LIN {X -0.022,Y -551.282,Z 288.033,A 0.000,B 0.000,C 90.000,E1 221.881} C_DIS
LIN {X -0.166,Y -545.235,Z 288.022,A 0.000,B 0.000,C 90.000,E1 219.930} C_DIS
LIN {X -0.082,Y -540.917,Z 288.014,A 0.000,B 0.000,C 90.000,E1 218.508} C_DIS
LIN {X 0.010,Y -536.637,Z 288.006,A 0.000,B 0.000,C 90.000,E1 217.076} C_DIS
LIN {X -0.298,Y -530.712,Z 287.995,A 0.000,B 0.000,C 90.000,E1 215.105} C_DIS
LIN {X 0.124,Y -524.882,Z 287.984,A 0.000,B 0.000,C 90.000,E1 213.038} C_DIS
LIN {X 0.156,Y -517.882,Z 287.969,A 0.000,B 0.000,C 90.000,E1 210.413} C_DIS
LIN {X -0.211,Y -511.936,Z 287.956,A 0.000,B 0.000,C 90.000,E1 208.103} C_DIS
LIN {X -0.005,Y -505.662,Z 287.941,A 0.000,B 0.000,C 90.000,E1 205.412} C_DIS
LIN {X -0.124,Y -501.187,Z 287.930,A 0.000,B 0.000,C 90.000,E1 203.334} C_DIS
LIN {X -0.097,Y -496.953,Z 287.918,A 0.000,B 0.000,C 90.000,E1 201.227} C_DIS
LIN {X 0.055,Y -493.512,Z 287.908,A 0.000,B 0.000,C 90.000,E1 199.396} C_DIS
LIN {X -0.125,Y -489.341,Z 287.894,A 0.000,B 0.000,C 90.000,E1 196.985} C_DIS
LIN {X -0.107,Y -485.490,Z 287.881,A 0.000,B 0.000,C 90.000,E1 194.537} C_DIS
LIN {X 0.015,Y -482.002,Z 287.867,A 0.000,B 0.000,C 90.000,E1 192.063} C_DIS
LIN {X -0.021,Y -479.203,Z 287.855,A 0.000,B 0.000,C 90.000,E1 189.905} C_DIS
LIN {X -0.211,Y -476.723,Z 287.843,A 0.000,B 0.000,C 90.000,E1 187.757} C_DIS
LIN {X 0.179,Y -474.137,Z 287.829,A 0.000,B 0.000,C 90.000,E1 185.220} C_DIS
LIN {X 0.182,Y -471.554,Z 287.814,A 0.000,B 0.000,C 90.000,E1 182.407} C_DIS
LIN {X 0.049,Y -469.852,Z 287.801,A 0.000,B 0.000,C 90.000,E1 180.229} C_DIS
LIN {X -0.125,Y -468.633,Z 287.789,A 0.000,B 0.000,C 90.000,E1 178.051} C_DIS
LIN {X 0.163,Y -467.261,Z 287.770,A 0.000,B 0.000,C 90.000,E1 174.552} C_DIS
LIN {X 0.067,Y -466.887,Z 287.758,A 0.000,B 0.000,C 90.000,E1 172.356} C_DIS
LIN {X 0.114,Y -466.574,Z 287.742,A 0.000,B 0.000,C 90.000,E1 169.511} C_DIS
LIN {X -0.130,Y -466.836,Z 287.726,A 0.000,B 0.000,C 90.000,E1 166.700} C_DIS
LIN {X 0.160,Y -468.096,Z 287.707,A 0.000,B 0.000,C 90.000,E1 163.196} C_DIS
LIN {X 0.075,Y -470.064,Z 287.689,A 0.000,B 0.000,C 90.000,E1 160.061} C_DIS
LIN {X 0.258,Y -471.526,Z 287.679,A 0.000,B 0.000,C 90.000,E1 158.156} C_DIS
LIN {X 0.123,Y -474.366,Z 287.663,A 0.000,B 0.000,C 90.000,E1 155.357} C_DIS
LIN {X -0.198,Y -478.123,Z 287.646,A 0.000,B 0.000,C 90.000,E1 152.281} C_DIS
LIN {X 0.097,Y -481.402,Z 287.634,A 0.000,B 0.000,C 90.000,E1 150.078} C_DIS
LIN {X 0.128,Y -484.933,Z 287.622,A 0.000,B 0.000,C 90.000,E1 147.916} C_DIS
LIN {X -0.149,Y -488.614,Z 287.610,A 0.000,B 0.000,C 90.000,E1 145.801} C_DIS
LIN {X -0.316,Y -491.783,Z 287.600,A 0.000,B 0.000,C 90.000,E1 143.989} C_DIS
LIN {X 0.172,Y -494.913,Z 287.590,A 0.000,B 0.000,C 90.000,E1 142.110} C_DIS
LIN {X -0.080,Y -496.875,Z 287.583,A 0.000,B 0.000,C 90.000,E1 140.928} C_DIS
LIN {X 0.076,Y -498.689,Z 287.576,A 0.000,B 0.000,C 90.000,E1 139.703} C_DIS
LIN {X 0.195,Y -500.322,Z 287.570,A 0.000,B 0.000,C 90.000,E1 138.485} C_DIS
LIN {X -0.034,Y -501.602,Z 287.563,A 0.000,B 0.000,C 90.000,E1 137.310} C_DIS
LIN {X 0.042,Y -502.103,Z 287.560,A 0.000,B 0.000,C 90.000,E1 136.701} C_DIS
LIN {X -0.028,Y -502.598,Z 287.555,A 0.000,B 0.000,C 90.000,E1 135.810} C_DIS
LIN {X -0.091,Y -502.898,Z 287.550,A 0.000,B 0.000,C 90.000,E1 134.919} C_DIS
LIN {X 0.067,Y -502.896,Z 287.543,A 0.000,B 0.000,C 90.000,E1 133.704} C_DIS
LIN {X 0.001,Y -502.579,Z 287.538,A 0.000,B 0.000,C 90.000,E1 132.813} C_DIS
LIN {X -0.038,Y -502.029,Z 287.533,A 0.000,B 0.000,C 90.000,E1 131.919} C_DIS
LIN {X 0.129,Y -500.892,Z 287.526,A 0.000,B 0.000,C 90.000,E1 130.701} C_DIS
LIN {X 0.081,Y -499.879,Z 287.521,A 0.000,B 0.000,C 90.000,E1 129.806} C_DIS
LIN {X -0.104,Y -498.289,Z 287.515,A 0.000,B 0.000,C 90.000,E1 128.624} C_DIS
LIN {X 0.078,Y -496.609,Z 287.508,A 0.000,B 0.000,C 90.000,E1 127.397} C_DIS
LIN {X -0.165,Y -494.765,Z 287.501,A 0.000,B 0.000,C 90.000,E1 126.217} C_DIS
LIN {X -0.078,Y -492.159,Z 287.493,A 0.000,B 0.000,C 90.000,E1 124.692} C_DIS
LIN {X -0.037,Y -489.306,Z 287.484,A 0.000,B 0.000,C 90.000,E1 123.166} C_DIS
LIN {X -0.082,Y -485.832,Z 287.474,A 0.000,B 0.000,C 90.000,E1 121.337} C_DIS
LIN {X -0.241,Y -483.532,Z 287.467,A 0.000,B 0.000,C 90.000,E1 120.129} C_DIS
LIN {X -0.277,Y -479.342,Z 287.455,A 0.000,B 0.000,C 90.000,E1 117.975} C_DIS
LIN {X -0.162,Y -476.366,Z 287.447,A 0.000,B 0.000,C 90.000,E1 116.411} C_DIS
LIN {X -0.068,Y -473.881,Z 287.440,A 0.000,B 0.000,C 90.000,E1 115.155} C_DIS
LIN {X -0.004,Y -471.585,Z 287.433,A 0.000,B 0.000,C 90.000,E1 113.898} C_DIS
LIN {X -0.174,Y -466.921,Z 287.419,A 0.000,B 0.000,C 90.000,E1 111.408} C_DIS
LIN {X -0.099,Y -463.544,Z 287.408,A 0.000,B 0.000,C 90.000,E1 109.504} C_DIS
LIN {X -0.105,Y -460.881,Z 287.400,A 0.000,B 0.000,C 90.000,E1 107.928} C_DIS
LIN {X -0.145,Y -460.875,Z 287.400,A 0.000,B 0.000,C 90.000,E1 107.928} C_DIS
LIN {X -0.237,Y -467.713,Z 287.383,A 0.000,B 0.000,C 90.000,E1 104.954} C_DIS
LIN {X 0.187,Y -475.922,Z 287.357,A 0.000,B 0.000,C 90.000,E1 100.197} C_DIS
LIN {X 0.027,Y -476.358,Z 287.355,A 0.000,B 0.000,C 90.000,E1 99.905} C_DIS
LIN {X -0.017,Y -481.880,Z 287.331,A 0.000,B 0.000,C 90.000,E1 95.568} C_DIS
LIN {X -0.170,Y -482.194,Z 287.329,A 0.000,B 0.000,C 90.000,E1 95.277} C_DIS
LIN {X -0.236,Y -485.368,Z 287.305,A 0.000,B 0.000,C 90.000,E1 90.974} C_DIS
LIN {X 0.073,Y -485.531,Z 287.304,A 0.000,B 0.000,C 90.000,E1 90.630} C_DIS
LIN {X -0.204,Y -486.347,Z 287.281,A 0.000,B 0.000,C 90.000,E1 86.674} C_DIS
LIN {X 0.106,Y -486.369,Z 287.280,A 0.000,B 0.000,C 90.000,E1 86.331} C_DIS
LIN {X -0.212,Y -486.061,Z 287.276,A 0.000,B 0.000,C 90.000,E1 85.755} C_DIS
LIN {X 0.130,Y -484.693,Z 287.254,A 0.000,B 0.000,C 90.000,E1 81.724} C_DIS
LIN {X -0.002,Y -484.531,Z 287.252,A 0.000,B 0.000,C 90.000,E1 81.432} C_DIS
LIN {X -0.132,Y -480.469,Z 287.227,A 0.000,B 0.000,C 90.000,E1 76.825} C_DIS
LIN {X -0.235,Y -474.228,Z 287.201,A 0.000,B 0.000,C 90.000,E1 72.181} C_DIS
LIN {X 0.183,Y -473.729,Z 287.199,A 0.000,B 0.000,C 90.000,E1 71.819} C_DIS
LIN {X 0.081,Y -472.855,Z 287.197,A 0.000,B 0.000,C 90.000,E1 71.402} C_DIS
LIN {X 0.041,Y -472.855,Z 287.197,A 0.000,B 0.000,C 90.000,E1 71.402} C_DIS
LIN {X 0.283,Y -476.430,Z 287.189,A 0.000,B 0.000,C 90.000,E1 69.934} C_DIS
LIN {X 0.008,Y -482.896,Z 287.175,A 0.000,B 0.000,C 90.000,E1 67.486} C_DIS
LIN {X -0.165,Y -489.519,Z 287.161,A 0.000,B 0.000,C 90.000,E1 65.049} C_DIS
LIN {X -0.053,Y -493.811,Z 287.153,A 0.000,B 0.000,C 90.000,E1 63.512} C_DIS
LIN {X -0.125,Y -500.706,Z 287.139,A 0.000,B 0.000,C 90.000,E1 61.101} C_DIS
LIN {X 0.059,Y -505.947,Z 287.129,A 0.000,B 0.000,C 90.000,E1 59.282} C_DIS
LIN {X 0.070,Y -512.082,Z 287.118,A 0.000,B 0.000,C 90.000,E1 57.199} C_DIS
LIN {X 0.086,Y -516.294,Z 287.110,A 0.000,B 0.000,C 90.000,E1 55.722} C_DIS
LIN {X -0.049,Y -519.604,Z 287.103,A 0.000,B 0.000,C 90.000,E1 54.562} C_DIS
LIN {X -0.263,Y -522.649,Z 287.097,A 0.000,B 0.000,C 90.000,E1 53.417} C_DIS
LIN {X 0.304,Y -525.486,Z 287.090,A 0.000,B 0.000,C 90.000,E1 52.190} C_DIS
LIN {X 0.203,Y -527.474,Z 287.085,A 0.000,B 0.000,C 90.000,E1 51.331} C_DIS
LIN {X 0.020,Y -529.949,Z 287.079,A 0.000,B 0.000,C 90.000,E1 50.194} C_DIS
LIN {X 0.301,Y -531.668,Z 287.074,A 0.000,B 0.000,C 90.000,E1 49.299} C_DIS
LIN {X -0.155,Y -533.178,Z 287.069,A 0.000,B 0.000,C 90.000,E1 48.485} C_DIS
LIN {X 0.102,Y -534.990,Z 287.063,A 0.000,B 0.000,C 90.000,E1 47.310} C_DIS
LIN {X 0.001,Y -536.441,Z 287.057,A 0.000,B 0.000,C 90.000,E1 46.176} C_DIS
LIN {X -0.070,Y -537.575,Z 287.050,A 0.000,B 0.000,C 90.000,E1 45.040} C_DIS
LIN {X 0.246,Y -538.429,Z 287.044,A 0.000,B 0.000,C 90.000,E1 43.866} C_DIS
LIN {X -0.179,Y -539.008,Z 287.038,A 0.000,B 0.000,C 90.000,E1 42.771} C_DIS
LIN {X 0.163,Y -539.340,Z 287.031,A 0.000,B 0.000,C 90.000,E1 41.595} C_DIS
LIN {X 0.149,Y -539.479,Z 287.025,A 0.000,B 0.000,C 90.000,E1 40.458} C_DIS
LIN {X -0.209,Y -539.367,Z 287.019,A 0.000,B 0.000,C 90.000,E1 39.358} C_DIS
LIN {X 0.209,Y -538.800,Z 287.011,A 0.000,B 0.000,C 90.000,E1 37.890} C_DIS
LIN {X -0.148,Y -537.903,Z 287.003,A 0.000,B 0.000,C 90.000,E1 36.503} C_DIS
LIN {X -0.107,Y -537.027,Z 286.996,A 0.000,B 0.000,C 90.000,E1 35.358} C_DIS
LIN {X 0.051,Y -535.988,Z 286.990,A 0.000,B 0.000,C 90.000,E1 34.199} C_DIS
LIN {X 0.193,Y -534.349,Z 286.981,A 0.000,B 0.000,C 90.000,E1 32.467} C_DIS
LIN {X -0.277,Y -532.519,Z 286.971,A 0.000,B 0.000,C 90.000,E1 30.797} C_DIS
LIN {X 0.141,Y -530.682,Z 286.961,A 0.000,B 0.000,C 90.000,E1 29.027} C_DIS
LIN {X 0.046,Y -528.801,Z 286.952,A 0.000,B 0.000,C 90.000,E1 27.308} C_DIS
LIN {X -0.114,Y -526.875,Z 286.942,A 0.000,B 0.000,C 90.000,E1 25.591} C_DIS
LIN {X 0.165,Y -525.172,Z 286.932,A 0.000,B 0.000,C 90.000,E1 23.823} C_DIS
LIN {X 0.157,Y -523.230,Z 286.921,A 0.000,B 0.000,C 90.000,E1 21.791} C_DIS
LIN {X -0.022,Y -521.984,Z 286.913,A 0.000,B 0.000,C 90.000,E1 20.355} C_DIS
LIN {X -0.103,Y -520.900,Z 286.905,A 0.000,B 0.000,C 90.000,E1 18.906} C_DIS
LIN {X -0.060,Y -519.660,Z 286.895,A 0.000,B 0.000,C 90.000,E1 17.149} C_DIS
LIN {X -0.251,Y -518.083,Z 286.881,A 0.000,B 0.000,C 90.000,E1 14.537} C_DIS
LIN {X -0.203,Y -517.233,Z 286.869,A 0.000,B 0.000,C 90.000,E1 12.479} C_DIS
LIN {X 0.189,Y -516.314,Z 286.853,A 0.000,B 0.000,C 90.000,E1 9.500} C_DIS
LIN {X -0.015,Y -516.024,Z 286.842,A 0.000,B 0.000,C 90.000,E1 7.466} C_DIS
LIN {X 0.141,Y -516.118,Z 286.830,A 0.000,B 0.000,C 90.000,E1 5.391} C_DIS
LIN {X -0.225,Y -516.505,Z 286.820,A 0.000,B 0.000,C 90.000,E1 3.669} C_DIS
LIN {X 0.127,Y -517.693,Z 286.802,A 0.000,B 0.000,C 90.000,E1 0.401} C_DIS
LIN {X -0.102,Y -519.014,Z 286.791,A 0.000,B 0.000,C 90.000,E1 358.339} C_DIS
LIN {X 0.061,Y -520.698,Z 286.779,A 0.000,B 0.000,C 90.000,E1 356.274} C_DIS
LIN {X 0.248,Y -523.662,Z 286.763,A 0.000,B 0.000,C 90.000,E1 353.337} C_DIS
LIN {X 0.219,Y -528.870,Z 286.744,A 0.000,B 0.000,C 90.000,E1 349.859} C_DIS
LIN {X -0.151,Y -533.012,Z 286.733,A 0.000,B 0.000,C 90.000,E1 347.881} C_DIS
LIN {X -0.010,Y -538.644,Z 286.720,A 0.000,B 0.000,C 90.000,E1 345.574} C_DIS
LIN {X 0.005,Y -542.943,Z 286.710,A 0.000,B 0.000,C 90.000,E1 343.866} C_DIS
LIN {X 0.036,Y -550.760,Z 286.695,A 0.000,B 0.000,C 90.000,E1 341.040} C_DIS
LIN {X 0.290,Y -561.382,Z 286.676,A 0.000,B 0.000,C 90.000,E1 337.667} C_DIS
LIN {X 0.104,Y -566.038,Z 286.668,A 0.000,B 0.000,C 90.000,E1 336.305} C_DIS
LIN {X 0.063,Y -568.796,Z 286.664,A 0.000,B 0.000,C 90.000,E1 335.485} C_DIS
LIN {X -0.284,Y -573.663,Z 286.656,A 0.000,B 0.000,C 90.000,E1 334.152} C_DIS
LIN {X 0.224,Y -578.648,Z 286.649,A 0.000,B 0.000,C 90.000,E1 332.743} C_DIS
LIN {X 0.175,Y -584.349,Z 286.640,A 0.000,B 0.000,C 90.000,E1 331.129} C_DIS
LIN {X 0.078,Y -587.101,Z 286.635,A 0.000,B 0.000,C 90.000,E1 330.333} C_DIS
LIN {X 0.173,Y -593.390,Z 286.625,A 0.000,B 0.000,C 90.000,E1 328.456} C_DIS
LIN {X -0.085,Y -599.852,Z 286.615,A 0.000,B 0.000,C 90.000,E1 326.628} C_DIS
LIN {X 0.137,Y -606.584,Z 286.604,A 0.000,B 0.000,C 90.000,E1 324.769} C_DIS
LIN {X -0.200,Y -611.352,Z 286.597,A 0.000,B 0.000,C 90.000,E1 323.497} C_DIS
LIN {X 0.098,Y -614.969,Z 286.591,A 0.000,B 0.000,C 90.000,E1 322.431} C_DIS
LIN {X -0.043,Y -618.442,Z 286.586,A 0.000,B 0.000,C 90.000,E1 321.412} C_DIS
LIN {X 0.022,Y -623.383,Z 286.577,A 0.000,B 0.000,C 90.000,E1 319.865} C_DIS
LIN {X 0.117,Y -628.029,Z 286.569,A 0.000,B 0.000,C 90.000,E1 318.324} C_DIS
LIN {X 0.083,Y -630.918,Z 286.563,A 0.000,B 0.000,C 90.000,E1 317.310} C_DIS
LIN {X -0.125,Y -635.283,Z 286.555,A 0.000,B 0.000,C 90.000,E1 315.810} C_DIS
LIN {X 0.290,Y -638.880,Z 286.547,A 0.000,B 0.000,C 90.000,E1 314.514} C_DIS
LIN {X -0.145,Y -642.391,Z 286.541,A 0.000,B 0.000,C 90.000,E1 313.299} C_DIS
LIN {X 0.088,Y -644.386,Z 286.536,A 0.000,B 0.000,C 90.000,E1 312.528} C_DIS
LIN {X 0.272,Y -646.963,Z 286.531,A 0.000,B 0.000,C 90.000,E1 311.515} C_DIS
LIN {X 0.060,Y -649.243,Z 286.525,A 0.000,B 0.000,C 90.000,E1 310.539} C_DIS
LIN {X -0.120,Y -651.334,Z 286.520,A 0.000,B 0.000,C 90.000,E1 309.564} C_DIS
LIN {X -0.298,Y -654.019,Z 286.512,A 0.000,B 0.000,C 90.000,E1 308.096} C_DIS
LIN {X 0.088,Y -655.509,Z 286.506,A 0.000,B 0.000,C 90.000,E1 307.076} C_DIS
LIN {X 0.102,Y -656.775,Z 286.501,A 0.000,B 0.000,C 90.000,E1 306.091} C_DIS
LIN {X 0.116,Y -657.281,Z 286.498,A 0.000,B 0.000,C 90.000,E1 305.598} C_DIS
LIN {X 0.154,Y -657.718,Z 286.492,A 0.000,B 0.000,C 90.000,E1 304.612} C_DIS
LIN {X 0.191,Y -657.885,Z 286.487,A 0.000,B 0.000,C 90.000,E1 303.627} C_DIS
LIN {X 0.310,Y -657.889,Z 286.483,A 0.000,B 0.000,C 90.000,E1 302.880} C_DIS
LIN {X 0.080,Y -657.516,Z 286.479,A 0.000,B 0.000,C 90.000,E1 302.163} C_DIS
LIN {X 0.091,Y -657.134,Z 286.476,A 0.000,B 0.000,C 90.000,E1 301.671} C_DIS
LIN {X 0.203,Y -656.212,Z 286.472,A 0.000,B 0.000,C 90.000,E1 300.924} C_DIS
LIN {X -0.030,Y -654.993,Z 286.468,A 0.000,B 0.000,C 90.000,E1 300.207} C_DIS
LIN {X 0.160,Y -652.992,Z 286.462,A 0.000,B 0.000,C 90.000,E1 299.205} C_DIS
LIN {X 0.001,Y -650.651,Z 286.457,A 0.000,B 0.000,C 90.000,E1 298.231} C_DIS
LIN {X -0.280,Y -648.844,Z 286.453,A 0.000,B 0.000,C 90.000,E1 297.513} C_DIS
LIN {X 0.170,Y -645.743,Z 286.446,A 0.000,B 0.000,C 90.000,E1 296.232} C_DIS
LIN {X -0.221,Y -641.747,Z 286.438,A 0.000,B 0.000,C 90.000,E1 294.771} C_DIS
LIN {X -0.166,Y -638.308,Z 286.431,A 0.000,B 0.000,C 90.000,E1 293.515} C_DIS
LIN {X -0.217,Y -635.664,Z 286.425,A 0.000,B 0.000,C 90.000,E1 292.514} C_DIS
LIN {X -0.102,Y -631.085,Z 286.415,A 0.000,B 0.000,C 90.000,E1 290.737} C_DIS
LIN {X -0.304,Y -625.969,Z 286.404,A 0.000,B 0.000,C 90.000,E1 288.725} C_DIS
LIN {X -0.035,Y -621.828,Z 286.394,A 0.000,B 0.000,C 90.000,E1 286.913} C_DIS
LIN {X 0.083,Y -617.059,Z 286.381,A 0.000,B 0.000,C 90.000,E1 284.592} C_DIS
LIN {X -0.023,Y -611.498,Z 286.362,A 0.000,B 0.000,C 90.000,E1 281.243} C_DIS
LIN {X 0.188,Y -608.186,Z 286.348,A 0.000,B 0.000,C 90.000,E1 278.624} C_DIS
LIN {X -0.246,Y -605.664,Z 286.332,A 0.000,B 0.000,C 90.000,E1 275.796} C_DIS
LIN {X -0.110,Y -604.050,Z 286.312,A 0.000,B 0.000,C 90.000,E1 272.121} C_DIS
LIN {X -0.009,Y -603.945,Z 286.294,A 0.000,B 0.000,C 90.000,E1 268.969} C_DIS
LIN {X -0.193,Y -605.476,Z 286.275,A 0.000,B 0.000,C 90.000,E1 265.584} C_DIS
LIN {X 0.194,Y -607.166,Z 286.264,A 0.000,B 0.000,C 90.000,E1 263.457} C_DIS
LIN {X 0.232,Y -610.043,Z 286.249,A 0.000,B 0.000,C 90.000,E1 260.849} C_DIS
LIN {X 0.136,Y -613.319,Z 286.236,A 0.000,B 0.000,C 90.000,E1 258.522} C_DIS
LIN {X 0.252,Y -616.132,Z 286.226,A 0.000,B 0.000,C 90.000,E1 256.700} C_DIS
LIN {X -0.173,Y -618.906,Z 286.216,A 0.000,B 0.000,C 90.000,E1 254.936} C_DIS
LIN {X -0.092,Y -619.987,Z 286.212,A 0.000,B 0.000,C 90.000,E1 254.157} C_DIS
LIN {X 0.005,Y -620.838,Z 286.208,A 0.000,B 0.000,C 90.000,E1 253.378} C_DIS
LIN {X 0.113,Y -621.447,Z 286.203,A 0.000,B 0.000,C 90.000,E1 252.598} C_DIS
LIN {X -0.248,Y -622.517,Z 286.195,A 0.000,B 0.000,C 90.000,E1 251.094} C_DIS
LIN {X -0.149,Y -622.786,Z 286.189,A 0.000,B 0.000,C 90.000,E1 250.061} C_DIS
LIN {X 0.181,Y -622.785,Z 286.185,A 0.000,B 0.000,C 90.000,E1 249.263} C_DIS
LIN {X -0.303,Y -622.345,Z 286.179,A 0.000,B 0.000,C 90.000,E1 248.284} C_DIS
LIN {X 0.019,Y -621.839,Z 286.175,A 0.000,B 0.000,C 90.000,E1 247.486} C_DIS
LIN {X -0.240,Y -621.023,Z 286.171,A 0.000,B 0.000,C 90.000,E1 246.741} C_DIS
LIN {X 0.301,Y -619.565,Z 286.165,A 0.000,B 0.000,C 90.000,E1 245.665} C_DIS
LIN {X 0.016,Y -618.228,Z 286.161,A 0.000,B 0.000,C 90.000,E1 244.921} C_DIS
LIN {X -0.038,Y -616.106,Z 286.155,A 0.000,B 0.000,C 90.000,E1 243.896} C_DIS
LIN {X -0.142,Y -613.014,Z 286.148,A 0.000,B 0.000,C 90.000,E1 242.615} C_DIS
LIN {X -0.015,Y -609.650,Z 286.141,A 0.000,B 0.000,C 90.000,E1 241.307} C_DIS
LIN {X 0.056,Y -606.046,Z 286.133,A 0.000,B 0.000,C 90.000,E1 239.999} C_DIS
LIN {X 0.120,Y -603.094,Z 286.128,A 0.000,B 0.000,C 90.000,E1 238.948} C_DIS
LIN {X 0.095,Y -598.460,Z 286.119,A 0.000,B 0.000,C 90.000,E1 237.375} C_DIS
LIN {X -0.239,Y -594.425,Z 286.112,A 0.000,B 0.000,C 90.000,E1 236.087} C_DIS
LIN {X 0.296,Y -591.080,Z 286.106,A 0.000,B 0.000,C 90.000,E1 234.975} C_DIS
LIN {X -0.124,Y -585.783,Z 286.097,A 0.000,B 0.000,C 90.000,E1 233.417} C_DIS
LIN {X -0.121,Y -579.944,Z 286.086,A 0.000,B 0.000,C 90.000,E1 231.537} C_DIS
LIN {X 0.084,Y -576.555,Z 286.080,A 0.000,B 0.000,C 90.000,E1 230.436} C_DIS
LIN {X 0.273,Y -569.783,Z 286.068,A 0.000,B 0.000,C 90.000,E1 228.243} C_DIS
LIN {X -0.035,Y -565.590,Z 286.061,A 0.000,B 0.000,C 90.000,E1 226.905} C_DIS
LIN {X 0.059,Y -560.458,Z 286.051,A 0.000,B 0.000,C 90.000,E1 225.243} C_DIS
LIN {X 0.043,Y -555.295,Z 286.042,A 0.000,B 0.000,C 90.000,E1 223.581} C_DIS
LIN {X -0.081,Y -550.166,Z 286.033,A 0.000,B 0.000,C 90.000,E1 221.919} C_DIS
LIN {X 0.112,Y -544.110,Z 286.022,A 0.000,B 0.000,C 90.000,E1 219.930} C_DIS
LIN {X -0.162,Y -539.773,Z 286.014,A 0.000,B 0.000,C 90.000,E1 218.543} C_DIS
LIN {X 0.243,Y -535.494,Z 286.006,A 0.000,B 0.000,C 90.000,E1 217.076} C_DIS
LIN {X -0.096,Y -529.555,Z 285.995,A 0.000,B 0.000,C 90.000,E1 215.105} C_DIS
LIN {X -0.145,Y -523.735,Z 285.984,A 0.000,B 0.000,C 90.000,E1 213.086} C_DIS
LIN {X 0.178,Y -517.508,Z 285.971,A 0.000,B 0.000,C 90.000,E1 210.718} C_DIS
LIN {X -0.117,Y -510.755,Z 285.956,A 0.000,B 0.000,C 90.000,E1 208.103} C_DIS
LIN {X 0.049,Y -504.490,Z 285.941,A 0.000,B 0.000,C 90.000,E1 205.412} C_DIS
LIN {X -0.173,Y -500.627,Z 285.931,A 0.000,B 0.000,C 90.000,E1 203.643} C_DIS
LIN {X -0.222,Y -496.967,Z 285.921,A 0.000,B 0.000,C 90.000,E1 201.844} C_DIS
LIN {X 0.023,Y -492.365,Z 285.908,A 0.000,B 0.000,C 90.000,E1 199.396} C_DIS
LIN {X -0.175,Y -487.682,Z 285.893,A 0.000,B 0.000,C 90.000,E1 196.677} C_DIS
LIN {X -0.206,Y -484.341,Z 285.881,A 0.000,B 0.000,C 90.000,E1 194.537} C_DIS
LIN {X 0.159,Y -481.701,Z 285.870,A 0.000,B 0.000,C 90.000,E1 192.647} C_DIS
LIN {X 0.112,Y -478.889,Z 285.858,A 0.000,B 0.000,C 90.000,E1 190.489} C_DIS
LIN {X -0.238,Y -475.986,Z 285.845,A 0.000,B 0.000,C 90.000,E1 188.049} C_DIS
LIN {X 0.137,Y -473.403,Z 285.831,A 0.000,B 0.000,C 90.000,E1 185.511} C_DIS
LIN {X 0.152,Y -470.823,Z 285.815,A 0.000,B 0.000,C 90.000,E1 182.694} C_DIS
LIN {X -0.231,Y -468.922,Z 285.801,A 0.000,B 0.000,C 90.000,E1 180.229} C_DIS
LIN {X 0.040,Y -467.675,Z 285.789,A 0.000,B 0.000,C 90.000,E1 177.993} C_DIS
LIN {X -0.150,Y -466.533,Z 285.773,A 0.000,B 0.000,C 90.000,E1 175.179} C_DIS
LIN {X -0.101,Y -466.011,Z 285.759,A 0.000,B 0.000,C 90.000,E1 172.648} C_DIS
LIN {X 0.107,Y -465.735,Z 285.745,A 0.000,B 0.000,C 90.000,E1 170.095} C_DIS
LIN {X 0.094,Y -465.947,Z 285.728,A 0.000,B 0.000,C 90.000,E1 166.937} C_DIS
LIN {X -0.234,Y -467.081,Z 285.708,A 0.000,B 0.000,C 90.000,E1 163.504} C_DIS
LIN {X 0.074,Y -469.009,Z 285.691,A 0.000,B 0.000,C 90.000,E1 160.315} C_DIS
LIN {X 0.180,Y -470.706,Z 285.679,A 0.000,B 0.000,C 90.000,E1 158.103} C_DIS
LIN {X 0.007,Y -473.564,Z 285.663,A 0.000,B 0.000,C 90.000,E1 155.305} C_DIS
LIN {X 0.028,Y -478.249,Z 285.642,A 0.000,B 0.000,C 90.000,E1 151.563} C_DIS
LIN {X -0.059,Y -481.117,Z 285.632,A 0.000,B 0.000,C 90.000,E1 149.715} C_DIS
LIN {X -0.090,Y -484.126,Z 285.621,A 0.000,B 0.000,C 90.000,E1 147.867} C_DIS
LIN {X -0.126,Y -487.808,Z 285.610,A 0.000,B 0.000,C 90.000,E1 145.722} C_DIS
LIN {X 0.090,Y -490.967,Z 285.599,A 0.000,B 0.000,C 90.000,E1 143.863} C_DIS
LIN {X -0.138,Y -494.100,Z 285.589,A 0.000,B 0.000,C 90.000,E1 142.065} C_DIS
LIN {X 0.289,Y -496.032,Z 285.582,A 0.000,B 0.000,C 90.000,E1 140.803} C_DIS
LIN {X 0.048,Y -497.847,Z 285.576,A 0.000,B 0.000,C 90.000,E1 139.622} C_DIS
LIN {X 0.155,Y -499.455,Z 285.569,A 0.000,B 0.000,C 90.000,E1 138.405} C_DIS
LIN {X -0.290,Y -500.456,Z 285.564,A 0.000,B 0.000,C 90.000,E1 137.553} C_DIS
LIN {X -0.016,Y -501.213,Z 285.559,A 0.000,B 0.000,C 90.000,E1 136.620} C_DIS
LIN {X -0.096,Y -501.697,Z 285.554,A 0.000,B 0.000,C 90.000,E1 135.729} C_DIS
LIN {X -0.168,Y -501.992,Z 285.549,A 0.000,B 0.000,C 90.000,E1 134.838} C_DIS
LIN {X -0.025,Y -501.965,Z 285.542,A 0.000,B 0.000,C 90.000,E1 133.623} C_DIS
LIN {X 0.267,Y -501.641,Z 285.537,A 0.000,B 0.000,C 90.000,E1 132.690} C_DIS
LIN {X -0.152,Y -501.077,Z 285.532,A 0.000,B 0.000,C 90.000,E1 131.838} C_DIS
LIN {X 0.129,Y -500.262,Z 285.527,A 0.000,B 0.000,C 90.000,E1 130.906} C_DIS
LIN {X 0.070,Y -499.291,Z 285.522,A 0.000,B 0.000,C 90.000,E1 130.011} C_DIS
LIN {X 0.002,Y -498.159,Z 285.517,A 0.000,B 0.000,C 90.000,E1 129.116} C_DIS
LIN {X 0.043,Y -496.109,Z 285.509,A 0.000,B 0.000,C 90.000,E1 127.604} C_DIS
LIN {X 0.191,Y -494.281,Z 285.502,A 0.000,B 0.000,C 90.000,E1 126.377} C_DIS
LIN {X 0.017,Y -492.225,Z 285.496,A 0.000,B 0.000,C 90.000,E1 125.185} C_DIS
LIN {X -0.187,Y -490.032,Z 285.489,A 0.000,B 0.000,C 90.000,E1 123.992} C_DIS
LIN {X 0.048,Y -486.552,Z 285.479,A 0.000,B 0.000,C 90.000,E1 122.133} C_DIS
LIN {X 0.102,Y -483.116,Z 285.468,A 0.000,B 0.000,C 90.000,E1 120.285} C_DIS
LIN {X 0.087,Y -479.531,Z 285.458,A 0.000,B 0.000,C 90.000,E1 118.437} C_DIS
LIN {X -0.242,Y -476.000,Z 285.448,A 0.000,B 0.000,C 90.000,E1 116.616} C_DIS
LIN {X 0.019,Y -472.919,Z 285.439,A 0.000,B 0.000,C 90.000,E1 115.027} C_DIS
LIN {X 0.068,Y -470.623,Z 285.432,A 0.000,B 0.000,C 90.000,E1 113.770} C_DIS
LIN {X -0.079,Y -466.530,Z 285.420,A 0.000,B 0.000,C 90.000,E1 111.589} C_DIS
LIN {X -0.239,Y -462.620,Z 285.408,A 0.000,B 0.000,C 90.000,E1 109.396} C_DIS
LIN {X -0.172,Y -460.487,Z 285.401,A 0.000,B 0.000,C 90.000,E1 108.127} C_DIS
LIN {X -0.068,Y -460.488,Z 285.401,A 0.000,B 0.000,C 90.000,E1 108.109} C_DIS
LIN {X -0.178,Y -467.240,Z 285.384,A 0.000,B 0.000,C 90.000,E1 105.134} C_DIS
LIN {X 0.199,Y -467.946,Z 285.382,A 0.000,B 0.000,C 90.000,E1 104.773} C_DIS
LIN {X 0.163,Y -476.164,Z 285.356,A 0.000,B 0.000,C 90.000,E1 100.074} C_DIS
LIN {X -0.106,Y -482.073,Z 285.330,A 0.000,B 0.000,C 90.000,E1 95.454} C_DIS
LIN {X 0.170,Y -485.496,Z 285.305,A 0.000,B 0.000,C 90.000,E1 90.802} C_DIS
LIN {X 0.202,Y -486.385,Z 285.281,A 0.000,B 0.000,C 90.000,E1 86.502} C_DIS
LIN {X 0.026,Y -486.362,Z 285.279,A 0.000,B 0.000,C 90.000,E1 86.216} C_DIS
LIN {X 0.109,Y -484.688,Z 285.253,A 0.000,B 0.000,C 90.000,E1 81.602} C_DIS
LIN {X 0.009,Y -480.613,Z 285.228,A 0.000,B 0.000,C 90.000,E1 76.992} C_DIS
LIN {X -0.132,Y -480.264,Z 285.226,A 0.000,B 0.000,C 90.000,E1 76.700} C_DIS
LIN {X 0.224,Y -474.091,Z 285.200,A 0.000,B 0.000,C 90.000,E1 72.000} C_DIS
LIN {X 0.092,Y -472.498,Z 285.196,A 0.000,B 0.000,C 90.000,E1 71.221} C_DIS
LIN {X 0.052,Y -472.508,Z 285.196,A 0.000,B 0.000,C 90.000,E1 71.221} C_DIS
LIN {X 0.124,Y -475.954,Z 285.188,A 0.000,B 0.000,C 90.000,E1 69.826} C_DIS
LIN {X 0.006,Y -481.581,Z 285.176,A 0.000,B 0.000,C 90.000,E1 67.667} C_DIS
LIN {X 0.217,Y -486.519,Z 285.166,A 0.000,B 0.000,C 90.000,E1 65.793} C_DIS
LIN {X -0.109,Y -492.490,Z 285.154,A 0.000,B 0.000,C 90.000,E1 63.691} C_DIS
LIN {X -0.014,Y -499.354,Z 285.140,A 0.000,B 0.000,C 90.000,E1 61.257} C_DIS
LIN {X 0.081,Y -503.715,Z 285.132,A 0.000,B 0.000,C 90.000,E1 59.744} C_DIS
LIN {X -0.289,Y -508.981,Z 285.122,A 0.000,B 0.000,C 90.000,E1 57.995} C_DIS
LIN {X -0.097,Y -512.459,Z 285.115,A 0.000,B 0.000,C 90.000,E1 56.786} C_DIS
LIN {X -0.071,Y -516.668,Z 285.107,A 0.000,B 0.000,C 90.000,E1 55.308} C_DIS
LIN {X 0.158,Y -519.117,Z 285.102,A 0.000,B 0.000,C 90.000,E1 54.402} C_DIS
LIN {X -0.105,Y -522.867,Z 285.094,A 0.000,B 0.000,C 90.000,E1 52.970} C_DIS
LIN {X -0.269,Y -525.631,Z 285.088,A 0.000,B 0.000,C 90.000,E1 51.823} C_DIS
LIN {X -0.097,Y -528.759,Z 285.080,A 0.000,B 0.000,C 90.000,E1 50.356} C_DIS
LIN {X 0.145,Y -531.038,Z 285.073,A 0.000,B 0.000,C 90.000,E1 49.175} C_DIS
LIN {X 0.012,Y -532.987,Z 285.067,A 0.000,B 0.000,C 90.000,E1 48.038} C_DIS
LIN {X 0.281,Y -534.281,Z 285.062,A 0.000,B 0.000,C 90.000,E1 47.148} C_DIS
LIN {X 0.205,Y -535.369,Z 285.057,A 0.000,B 0.000,C 90.000,E1 46.296} C_DIS
LIN {X 0.110,Y -536.541,Z 285.051,A 0.000,B 0.000,C 90.000,E1 45.162} C_DIS
LIN {X 0.022,Y -537.554,Z 285.043,A 0.000,B 0.000,C 90.000,E1 43.743} C_DIS
LIN {X -0.045,Y -538.094,Z 285.037,A 0.000,B 0.000,C 90.000,E1 42.609} C_DIS
LIN {X -0.075,Y -538.421,Z 285.030,A 0.000,B 0.000,C 90.000,E1 41.472} C_DIS
LIN {X -0.097,Y -538.472,Z 285.024,A 0.000,B 0.000,C 90.000,E1 40.334} C_DIS
LIN {X -0.134,Y -538.371,Z 285.019,A 0.000,B 0.000,C 90.000,E1 39.483} C_DIS
LIN {X 0.259,Y -537.809,Z 285.011,A 0.000,B 0.000,C 90.000,E1 38.016} C_DIS
LIN {X 0.312,Y -536.916,Z 285.003,A 0.000,B 0.000,C 90.000,E1 36.583} C_DIS
LIN {X 0.029,Y -536.055,Z 284.997,A 0.000,B 0.000,C 90.000,E1 35.471} C_DIS
LIN {X 0.044,Y -535.005,Z 284.991,A 0.000,B 0.000,C 90.000,E1 34.326} C_DIS
LIN {X 0.170,Y -533.593,Z 284.983,A 0.000,B 0.000,C 90.000,E1 32.880} C_DIS
LIN {X -0.016,Y -532.090,Z 284.975,A 0.000,B 0.000,C 90.000,E1 31.465} C_DIS
LIN {X 0.226,Y -530.515,Z 284.967,A 0.000,B 0.000,C 90.000,E1 30.001} C_DIS
LIN {X 0.131,Y -528.653,Z 284.957,A 0.000,B 0.000,C 90.000,E1 28.281} C_DIS
LIN {X -0.033,Y -526.727,Z 284.948,A 0.000,B 0.000,C 90.000,E1 26.565} C_DIS
LIN {X 0.010,Y -524.021,Z 284.933,A 0.000,B 0.000,C 90.000,E1 23.951} C_DIS
LIN {X 0.168,Y -522.045,Z 284.922,A 0.000,B 0.000,C 90.000,E1 21.897} C_DIS
LIN {X -0.072,Y -520.517,Z 284.912,A 0.000,B 0.000,C 90.000,E1 20.174} C_DIS
LIN {X -0.152,Y -519.644,Z 284.906,A 0.000,B 0.000,C 90.000,E1 19.014} C_DIS
LIN {X 0.195,Y -518.388,Z 284.896,A 0.000,B 0.000,C 90.000,E1 17.221} C_DIS
LIN {X 0.107,Y -516.751,Z 284.881,A 0.000,B 0.000,C 90.000,E1 14.592} C_DIS
LIN {X 0.116,Y -515.849,Z 284.870,A 0.000,B 0.000,C 90.000,E1 12.535} C_DIS
LIN {X -0.038,Y -514.972,Z 284.855,A 0.000,B 0.000,C 90.000,E1 9.905} C_DIS
LIN {X 0.140,Y -514.576,Z 284.842,A 0.000,B 0.000,C 90.000,E1 7.530} C_DIS
LIN {X 0.240,Y -514.666,Z 284.829,A 0.000,B 0.000,C 90.000,E1 5.163} C_DIS
LIN {X -0.153,Y -515.029,Z 284.819,A 0.000,B 0.000,C 90.000,E1 3.440} C_DIS
LIN {X 0.144,Y -516.265,Z 284.801,A 0.000,B 0.000,C 90.000,E1 0.172} C_DIS
LIN {X -0.178,Y -517.654,Z 284.789,A 0.000,B 0.000,C 90.000,E1 358.051} C_DIS
LIN {X -0.072,Y -519.389,Z 284.778,A 0.000,B 0.000,C 90.000,E1 355.988} C_DIS
LIN {X 0.055,Y -522.457,Z 284.761,A 0.000,B 0.000,C 90.000,E1 353.053} C_DIS
LIN {X -0.019,Y -526.277,Z 284.747,A 0.000,B 0.000,C 90.000,E1 350.443} C_DIS
LIN {X 0.129,Y -531.473,Z 284.732,A 0.000,B 0.000,C 90.000,E1 347.825} C_DIS
LIN {X 0.225,Y -537.118,Z 284.720,A 0.000,B 0.000,C 90.000,E1 345.519} C_DIS
LIN {X -0.100,Y -542.158,Z 284.709,A 0.000,B 0.000,C 90.000,E1 343.559} C_DIS
LIN {X -0.086,Y -550.124,Z 284.693,A 0.000,B 0.000,C 90.000,E1 340.732} C_DIS
LIN {X -0.160,Y -559.982,Z 284.676,A 0.000,B 0.000,C 90.000,E1 337.667} C_DIS
LIN {X -0.146,Y -564.659,Z 284.668,A 0.000,B 0.000,C 90.000,E1 336.282} C_DIS
LIN {X 0.300,Y -570.384,Z 284.659,A 0.000,B 0.000,C 90.000,E1 334.588} C_DIS
LIN {X -0.172,Y -576.353,Z 284.650,A 0.000,B 0.000,C 90.000,E1 332.999} C_DIS
LIN {X -0.130,Y -581.185,Z 284.642,A 0.000,B 0.000,C 90.000,E1 331.641} C_DIS
LIN {X 0.118,Y -584.928,Z 284.636,A 0.000,B 0.000,C 90.000,E1 330.539} C_DIS
LIN {X -0.035,Y -590.334,Z 284.628,A 0.000,B 0.000,C 90.000,E1 328.948} C_DIS
LIN {X 0.231,Y -595.801,Z 284.619,A 0.000,B 0.000,C 90.000,E1 327.327} C_DIS
LIN {X -0.144,Y -602.451,Z 284.608,A 0.000,B 0.000,C 90.000,E1 325.515} C_DIS
LIN {X 0.220,Y -608.292,Z 284.600,A 0.000,B 0.000,C 90.000,E1 323.909} C_DIS
LIN {X -0.005,Y -612.051,Z 284.594,A 0.000,B 0.000,C 90.000,E1 322.889} C_DIS
LIN {X -0.255,Y -616.443,Z 284.587,A 0.000,B 0.000,C 90.000,E1 321.618} C_DIS
LIN {X 0.332,Y -620.639,Z 284.580,A 0.000,B 0.000,C 90.000,E1 320.275} C_DIS
LIN {X -0.061,Y -623.061,Z 284.575,A 0.000,B 0.000,C 90.000,E1 319.542} C_DIS
LIN {X 0.036,Y -627.693,Z 284.567,A 0.000,B 0.000,C 90.000,E1 318.000} C_DIS
LIN {X 0.226,Y -632.056,Z 284.558,A 0.000,B 0.000,C 90.000,E1 316.458} C_DIS
LIN {X -0.315,Y -635.684,Z 284.551,A 0.000,B 0.000,C 90.000,E1 315.243} C_DIS
LIN {X 0.105,Y -639.240,Z 284.544,A 0.000,B 0.000,C 90.000,E1 313.947} C_DIS
LIN {X 0.140,Y -642.685,Z 284.537,A 0.000,B 0.000,C 90.000,E1 312.690} C_DIS
LIN {X -0.200,Y -645.841,Z 284.530,A 0.000,B 0.000,C 90.000,E1 311.472} C_DIS
LIN {X 0.001,Y -648.102,Z 284.525,A 0.000,B 0.000,C 90.000,E1 310.458} C_DIS
LIN {X -0.196,Y -650.120,Z 284.519,A 0.000,B 0.000,C 90.000,E1 309.483} C_DIS
LIN {X 0.070,Y -652.330,Z 284.512,A 0.000,B 0.000,C 90.000,E1 308.222} C_DIS
LIN {X 0.034,Y -653.874,Z 284.507,A 0.000,B 0.000,C 90.000,E1 307.237} C_DIS
LIN {X 0.030,Y -655.174,Z 284.501,A 0.000,B 0.000,C 90.000,E1 306.251} C_DIS
LIN {X 0.036,Y -655.707,Z 284.499,A 0.000,B 0.000,C 90.000,E1 305.758} C_DIS
LIN {X 0.059,Y -656.208,Z 284.493,A 0.000,B 0.000,C 90.000,E1 304.771} C_DIS
LIN {X 0.084,Y -656.399,Z 284.488,A 0.000,B 0.000,C 90.000,E1 303.785} C_DIS
LIN {X 0.191,Y -656.458,Z 284.484,A 0.000,B 0.000,C 90.000,E1 303.038} C_DIS
LIN {X -0.252,Y -656.133,Z 284.480,A 0.000,B 0.000,C 90.000,E1 302.339} C_DIS
LIN {X 0.303,Y -655.785,Z 284.477,A 0.000,B 0.000,C 90.000,E1 301.799} C_DIS
LIN {X 0.063,Y -654.943,Z 284.473,A 0.000,B 0.000,C 90.000,E1 301.082} C_DIS
LIN {X 0.153,Y -653.782,Z 284.469,A 0.000,B 0.000,C 90.000,E1 300.335} C_DIS
LIN {X 0.325,Y -651.822,Z 284.463,A 0.000,B 0.000,C 90.000,E1 299.333} C_DIS
LIN {X 0.053,Y -650.127,Z 284.459,A 0.000,B 0.000,C 90.000,E1 298.615} C_DIS
LIN {X -0.142,Y -647.721,Z 284.454,A 0.000,B 0.000,C 90.000,E1 297.641} C_DIS
LIN {X -0.212,Y -643.974,Z 284.445,A 0.000,B 0.000,C 90.000,E1 296.155} C_DIS
LIN {X 0.001,Y -639.276,Z 284.436,A 0.000,B 0.000,C 90.000,E1 294.387} C_DIS
LIN {X -0.154,Y -634.569,Z 284.426,A 0.000,B 0.000,C 90.000,E1 292.642} C_DIS
LIN {X -0.061,Y -629.958,Z 284.416,A 0.000,B 0.000,C 90.000,E1 290.865} C_DIS
LIN {X -0.086,Y -624.854,Z 284.405,A 0.000,B 0.000,C 90.000,E1 288.833} C_DIS
LIN {X -0.038,Y -620.684,Z 284.395,A 0.000,B 0.000,C 90.000,E1 287.040} C_DIS
LIN {X -0.177,Y -615.405,Z 284.380,A 0.000,B 0.000,C 90.000,E1 284.481} C_DIS
LIN {X -0.085,Y -610.286,Z 284.363,A 0.000,B 0.000,C 90.000,E1 281.366} C_DIS
LIN {X 0.103,Y -606.934,Z 284.349,A 0.000,B 0.000,C 90.000,E1 278.746} C_DIS
LIN {X 0.308,Y -604.379,Z 284.333,A 0.000,B 0.000,C 90.000,E1 275.853} C_DIS
LIN {X -0.126,Y -602.806,Z 284.315,A 0.000,B 0.000,C 90.000,E1 272.751} C_DIS
LIN {X -0.241,Y -602.479,Z 284.302,A 0.000,B 0.000,C 90.000,E1 270.401} C_DIS
LIN {X 0.075,Y -602.638,Z 284.293,A 0.000,B 0.000,C 90.000,E1 268.797} C_DIS
LIN {X -0.171,Y -604.244,Z 284.274,A 0.000,B 0.000,C 90.000,E1 265.412} C_DIS
LIN {X -0.112,Y -606.283,Z 284.261,A 0.000,B 0.000,C 90.000,E1 263.053} C_DIS
LIN {X -0.169,Y -608.653,Z 284.250,A 0.000,B 0.000,C 90.000,E1 260.971} C_DIS
LIN {X -0.204,Y -611.908,Z 284.237,A 0.000,B 0.000,C 90.000,E1 258.634} C_DIS
LIN {X -0.256,Y -614.759,Z 284.227,A 0.000,B 0.000,C 90.000,E1 256.825} C_DIS
LIN {X 0.032,Y -617.541,Z 284.217,A 0.000,B 0.000,C 90.000,E1 254.991} C_DIS
LIN {X 0.102,Y -618.646,Z 284.212,A 0.000,B 0.000,C 90.000,E1 254.212} C_DIS
LIN {X 0.011,Y -619.541,Z 284.208,A 0.000,B 0.000,C 90.000,E1 253.449} C_DIS
LIN {X 0.100,Y -620.187,Z 284.204,A 0.000,B 0.000,C 90.000,E1 252.670} C_DIS
LIN {X -0.096,Y -621.219,Z 284.195,A 0.000,B 0.000,C 90.000,E1 251.148} C_DIS
LIN {X -0.011,Y -621.533,Z 284.190,A 0.000,B 0.000,C 90.000,E1 250.115} C_DIS
LIN {X 0.090,Y -621.542,Z 284.185,A 0.000,B 0.000,C 90.000,E1 249.337} C_DIS
LIN {X -0.187,Y -621.154,Z 284.180,A 0.000,B 0.000,C 90.000,E1 248.337} C_DIS
LIN {X 0.118,Y -620.429,Z 284.174,A 0.000,B 0.000,C 90.000,E1 247.283} C_DIS
LIN {X -0.151,Y -619.503,Z 284.170,A 0.000,B 0.000,C 90.000,E1 246.538} C_DIS
LIN {X 0.133,Y -618.425,Z 284.165,A 0.000,B 0.000,C 90.000,E1 245.741} C_DIS
LIN {X 0.095,Y -617.083,Z 284.161,A 0.000,B 0.000,C 90.000,E1 244.973} C_DIS
LIN {X 0.029,Y -614.959,Z 284.155,A 0.000,B 0.000,C 90.000,E1 243.948} C_DIS
LIN {X -0.060,Y -612.521,Z 284.150,A 0.000,B 0.000,C 90.000,E1 242.922} C_DIS
LIN {X -0.186,Y -609.892,Z 284.144,A 0.000,B 0.000,C 90.000,E1 241.897} C_DIS
LIN {X -0.061,Y -607.130,Z 284.138,A 0.000,B 0.000,C 90.000,E1 240.845} C_DIS
LIN {X -0.035,Y -603.505,Z 284.131,A 0.000,B 0.000,C 90.000,E1 239.537} C_DIS
LIN {X 0.226,Y -599.708,Z 284.124,A 0.000,B 0.000,C 90.000,E1 238.201} C_DIS
LIN {X -0.089,Y -595.782,Z 284.116,A 0.000,B 0.000,C 90.000,E1 236.914} C_DIS
LIN {X -0.358,Y -592.518,Z 284.110,A 0.000,B 0.000,C 90.000,E1 235.881} C_DIS
LIN {X 0.150,Y -589.079,Z 284.104,A 0.000,B 0.000,C 90.000,E1 234.769} C_DIS
LIN {X 0.233,Y -581.335,Z 284.091,A 0.000,B 0.000,C 90.000,E1 232.351} C_DIS
LIN {X 0.166,Y -577.189,Z 284.084,A 0.000,B 0.000,C 90.000,E1 231.009} C_DIS
LIN {X 0.176,Y -572.051,Z 284.074,A 0.000,B 0.000,C 90.000,E1 229.380} C_DIS
LIN {X 0.019,Y -567.020,Z 284.065,A 0.000,B 0.000,C 90.000,E1 227.757} C_DIS
LIN {X 0.079,Y -562.781,Z 284.058,A 0.000,B 0.000,C 90.000,E1 226.377} C_DIS
LIN {X -0.292,Y -557.588,Z 284.049,A 0.000,B 0.000,C 90.000,E1 224.757} C_DIS
LIN {X -0.018,Y -553.298,Z 284.041,A 0.000,B 0.000,C 90.000,E1 223.338} C_DIS
LIN {X -0.187,Y -548.130,Z 284.031,A 0.000,B 0.000,C 90.000,E1 221.676} C_DIS
LIN {X -0.011,Y -542.936,Z 284.022,A 0.000,B 0.000,C 90.000,E1 219.967} C_DIS
LIN {X 0.041,Y -538.580,Z 284.014,A 0.000,B 0.000,C 90.000,E1 218.543} C_DIS
LIN {X -0.327,Y -534.302,Z 284.006,A 0.000,B 0.000,C 90.000,E1 217.156} C_DIS
LIN {X 0.053,Y -528.347,Z 283.995,A 0.000,B 0.000,C 90.000,E1 215.105} C_DIS
LIN {X -0.028,Y -522.552,Z 283.984,A 0.000,B 0.000,C 90.000,E1 213.086} C_DIS
LIN {X -0.007,Y -516.302,Z 283.971,A 0.000,B 0.000,C 90.000,E1 210.747} C_DIS
LIN {X -0.077,Y -509.539,Z 283.956,A 0.000,B 0.000,C 90.000,E1 208.103} C_DIS
LIN {X -0.033,Y -503.963,Z 283.943,A 0.000,B 0.000,C 90.000,E1 205.720} C_DIS
LIN {X 0.186,Y -500.094,Z 283.933,A 0.000,B 0.000,C 90.000,E1 203.898} C_DIS
LIN {X 0.127,Y -496.349,Z 283.923,A 0.000,B 0.000,C 90.000,E1 202.099} C_DIS
LIN {X -0.114,Y -493.987,Z 283.916,A 0.000,B 0.000,C 90.000,E1 200.918} C_DIS
LIN {X -0.030,Y -490.639,Z 283.906,A 0.000,B 0.000,C 90.000,E1 199.087} C_DIS
LIN {X 0.166,Y -486.545,Z 283.893,A 0.000,B 0.000,C 90.000,E1 196.622} C_DIS
LIN {X 0.106,Y -483.174,Z 283.881,A 0.000,B 0.000,C 90.000,E1 194.481} C_DIS
LIN {X 0.118,Y -480.995,Z 283.872,A 0.000,B 0.000,C 90.000,E1 192.939} C_DIS
LIN {X 0.051,Y -478.177,Z 283.860,A 0.000,B 0.000,C 90.000,E1 190.782} C_DIS
LIN {X -0.009,Y -474.916,Z 283.844,A 0.000,B 0.000,C 90.000,E1 187.992} C_DIS
LIN {X -0.137,Y -472.332,Z 283.831,A 0.000,B 0.000,C 90.000,E1 185.511} C_DIS
LIN {X -0.155,Y -469.822,Z 283.815,A 0.000,B 0.000,C 90.000,E1 182.694} C_DIS
LIN {X -0.098,Y -467.987,Z 283.801,A 0.000,B 0.000,C 90.000,E1 180.172} C_DIS
LIN {X -0.098,Y -466.907,Z 283.790,A 0.000,B 0.000,C 90.000,E1 178.282} C_DIS
LIN {X -0.095,Y -466.051,Z 283.780,A 0.000,B 0.000,C 90.000,E1 176.388} C_DIS
LIN {X 0.147,Y -465.256,Z 283.764,A 0.000,B 0.000,C 90.000,E1 173.514} C_DIS
LIN {X -0.196,Y -464.992,Z 283.754,A 0.000,B 0.000,C 90.000,E1 171.659} C_DIS
LIN {X 0.182,Y -464.853,Z 283.741,A 0.000,B 0.000,C 90.000,E1 169.398} C_DIS
LIN {X 0.235,Y -465.259,Z 283.724,A 0.000,B 0.000,C 90.000,E1 166.228} C_DIS
LIN {X 0.009,Y -466.546,Z 283.704,A 0.000,B 0.000,C 90.000,E1 162.779} C_DIS
LIN {X 0.125,Y -468.177,Z 283.690,A 0.000,B 0.000,C 90.000,E1 160.242} C_DIS
LIN {X 0.175,Y -470.216,Z 283.676,A 0.000,B 0.000,C 90.000,E1 157.720} C_DIS
LIN {X -0.009,Y -473.121,Z 283.661,A 0.000,B 0.000,C 90.000,E1 154.921} C_DIS
LIN {X -0.041,Y -478.436,Z 283.638,A 0.000,B 0.000,C 90.000,E1 150.873} C_DIS
LIN {X 0.106,Y -481.355,Z 283.628,A 0.000,B 0.000,C 90.000,E1 148.997} C_DIS
LIN {X 0.143,Y -484.900,Z 283.616,A 0.000,B 0.000,C 90.000,E1 146.834} C_DIS
LIN {X 0.069,Y -487.525,Z 283.607,A 0.000,B 0.000,C 90.000,E1 145.308} C_DIS
LIN {X 0.039,Y -490.161,Z 283.599,A 0.000,B 0.000,C 90.000,E1 143.783} C_DIS
LIN {X -0.053,Y -492.786,Z 283.590,A 0.000,B 0.000,C 90.000,E1 142.271} C_DIS
LIN {X 0.044,Y -494.735,Z 283.584,A 0.000,B 0.000,C 90.000,E1 141.045} C_DIS
LIN {X 0.101,Y -496.582,Z 283.577,A 0.000,B 0.000,C 90.000,E1 139.828} C_DIS
LIN {X 0.193,Y -498.229,Z 283.570,A 0.000,B 0.000,C 90.000,E1 138.609} C_DIS
LIN {X 0.308,Y -499.608,Z 283.564,A 0.000,B 0.000,C 90.000,E1 137.391} C_DIS
LIN {X -0.135,Y -500.328,Z 283.559,A 0.000,B 0.000,C 90.000,E1 136.539} C_DIS
LIN {X -0.225,Y -500.800,Z 283.553,A 0.000,B 0.000,C 90.000,E1 135.648} C_DIS
LIN {X 0.046,Y -501.087,Z 283.548,A 0.000,B 0.000,C 90.000,E1 134.717} C_DIS
LIN {X 0.323,Y -501.079,Z 283.543,A 0.000,B 0.000,C 90.000,E1 133.785} C_DIS
LIN {X -0.103,Y -500.850,Z 283.539,A 0.000,B 0.000,C 90.000,E1 132.933} C_DIS
LIN {X 0.178,Y -500.356,Z 283.534,A 0.000,B 0.000,C 90.000,E1 132.000} C_DIS
LIN {X -0.254,Y -499.609,Z 283.529,A 0.000,B 0.000,C 90.000,E1 131.148} C_DIS
LIN {X 0.006,Y -498.672,Z 283.523,A 0.000,B 0.000,C 90.000,E1 130.216} C_DIS
LIN {X -0.072,Y -497.579,Z 283.518,A 0.000,B 0.000,C 90.000,E1 129.322} C_DIS
LIN {X -0.045,Y -495.579,Z 283.510,A 0.000,B 0.000,C 90.000,E1 127.810} C_DIS
LIN {X 0.233,Y -494.266,Z 283.505,A 0.000,B 0.000,C 90.000,E1 126.870} C_DIS
LIN {X 0.058,Y -492.288,Z 283.498,A 0.000,B 0.000,C 90.000,E1 125.678} C_DIS
LIN {X -0.301,Y -489.586,Z 283.490,A 0.000,B 0.000,C 90.000,E1 124.199} C_DIS
LIN {X 0.099,Y -486.691,Z 283.481,A 0.000,B 0.000,C 90.000,E1 122.625} C_DIS
LIN {X 0.216,Y -482.669,Z 283.469,A 0.000,B 0.000,C 90.000,E1 120.463} C_DIS
LIN {X -0.023,Y -479.722,Z 283.461,A 0.000,B 0.000,C 90.000,E1 118.949} C_DIS
LIN {X 0.073,Y -476.161,Z 283.451,A 0.000,B 0.000,C 90.000,E1 117.078} C_DIS
LIN {X -0.050,Y -473.798,Z 283.444,A 0.000,B 0.000,C 90.000,E1 115.848} C_DIS
LIN {X 0.078,Y -469.651,Z 283.431,A 0.000,B 0.000,C 90.000,E1 113.643} C_DIS
LIN {X -0.097,Y -465.582,Z 283.419,A 0.000,B 0.000,C 90.000,E1 111.461} C_DIS
LIN {X 0.150,Y -461.685,Z 283.407,A 0.000,B 0.000,C 90.000,E1 109.214} C_DIS
LIN {X -0.072,Y -460.104,Z 283.402,A 0.000,B 0.000,C 90.000,E1 108.308} C_DIS
LIN {X -0.113,Y -460.101,Z 283.402,A 0.000,B 0.000,C 90.000,E1 108.308} C_DIS
LIN {X -0.245,Y -467.261,Z 283.384,A 0.000,B 0.000,C 90.000,E1 105.134} C_DIS
LIN {X 0.131,Y -467.958,Z 283.382,A 0.000,B 0.000,C 90.000,E1 104.773} C_DIS
LIN {X 0.094,Y -476.176,Z 283.356,A 0.000,B 0.000,C 90.000,E1 100.074} C_DIS
LIN {X -0.130,Y -482.084,Z 283.330,A 0.000,B 0.000,C 90.000,E1 95.448} C_DIS
LIN {X 0.100,Y -485.503,Z 283.305,A 0.000,B 0.000,C 90.000,E1 90.802} C_DIS
LIN {X 0.133,Y -486.384,Z 283.281,A 0.000,B 0.000,C 90.000,E1 86.502} C_DIS
LIN {X -0.043,Y -486.362,Z 283.279,A 0.000,B 0.000,C 90.000,E1 86.216} C_DIS
LIN {X 0.040,Y -484.686,Z 283.253,A 0.000,B 0.000,C 90.000,E1 81.602} C_DIS
LIN {X -0.060,Y -480.609,Z 283.228,A 0.000,B 0.000,C 90.000,E1 76.992} C_DIS
LIN {X -0.202,Y -480.249,Z 283.226,A 0.000,B 0.000,C 90.000,E1 76.700} C_DIS
LIN {X 0.154,Y -474.079,Z 283.200,A 0.000,B 0.000,C 90.000,E1 72.000} C_DIS
LIN {X 0.148,Y -472.156,Z 283.195,A 0.000,B 0.000,C 90.000,E1 71.040} C_DIS
LIN {X 0.108,Y -472.153,Z 283.195,A 0.000,B 0.000,C 90.000,E1 71.040} C_DIS
LIN {X 0.047,Y -475.198,Z 283.188,A 0.000,B 0.000,C 90.000,E1 69.826} C_DIS
LIN {X -0.092,Y -480.831,Z 283.176,A 0.000,B 0.000,C 90.000,E1 67.667} C_DIS
LIN {X 0.110,Y -486.568,Z 283.164,A 0.000,B 0.000,C 90.000,E1 65.485} C_DIS
LIN {X -0.046,Y -490.848,Z 283.155,A 0.000,B 0.000,C 90.000,E1 63.973} C_DIS
LIN {X -0.085,Y -495.929,Z 283.145,A 0.000,B 0.000,C 90.000,E1 62.153} C_DIS
LIN {X -0.004,Y -501.205,Z 283.135,A 0.000,B 0.000,C 90.000,E1 60.333} C_DIS
LIN {X 0.005,Y -506.418,Z 283.125,A 0.000,B 0.000,C 90.000,E1 58.535} C_DIS
LIN {X 0.162,Y -509.967,Z 283.119,A 0.000,B 0.000,C 90.000,E1 57.327} C_DIS
LIN {X -0.145,Y -514.221,Z 283.110,A 0.000,B 0.000,C 90.000,E1 55.881} C_DIS
LIN {X -0.016,Y -517.526,Z 283.104,A 0.000,B 0.000,C 90.000,E1 54.689} C_DIS
LIN {X 0.161,Y -520.580,Z 283.097,A 0.000,B 0.000,C 90.000,E1 53.497} C_DIS
LIN {X 0.008,Y -522.764,Z 283.092,A 0.000,B 0.000,C 90.000,E1 52.637} C_DIS
LIN {X 0.163,Y -525.487,Z 283.086,A 0.000,B 0.000,C 90.000,E1 51.457} C_DIS
LIN {X 0.025,Y -527.941,Z 283.080,A 0.000,B 0.000,C 90.000,E1 50.312} C_DIS
LIN {X -0.153,Y -530.212,Z 283.073,A 0.000,B 0.000,C 90.000,E1 49.175} C_DIS
LIN {X 0.057,Y -532.155,Z 283.067,A 0.000,B 0.000,C 90.000,E1 48.000} C_DIS
LIN {X -0.021,Y -533.030,Z 283.064,A 0.000,B 0.000,C 90.000,E1 47.433} C_DIS
LIN {X -0.105,Y -534.152,Z 283.059,A 0.000,B 0.000,C 90.000,E1 46.581} C_DIS
LIN {X -0.183,Y -535.085,Z 283.054,A 0.000,B 0.000,C 90.000,E1 45.729} C_DIS
LIN {X -0.235,Y -535.629,Z 283.051,A 0.000,B 0.000,C 90.000,E1 45.162} C_DIS
LIN {X 0.032,Y -536.605,Z 283.043,A 0.000,B 0.000,C 90.000,E1 43.704} C_DIS
LIN {X 0.339,Y -537.146,Z 283.037,A 0.000,B 0.000,C 90.000,E1 42.528} C_DIS
LIN {X -0.108,Y -537.469,Z 283.030,A 0.000,B 0.000,C 90.000,E1 41.434} C_DIS
LIN {X -0.152,Y -537.456,Z 283.024,A 0.000,B 0.000,C 90.000,E1 40.297} C_DIS
LIN {X -0.133,Y -537.322,Z 283.019,A 0.000,B 0.000,C 90.000,E1 39.439} C_DIS
LIN {X 0.231,Y -536.997,Z 283.014,A 0.000,B 0.000,C 90.000,E1 38.543} C_DIS
LIN {X -0.166,Y -536.546,Z 283.010,A 0.000,B 0.000,C 90.000,E1 37.729} C_DIS
LIN {X -0.136,Y -535.627,Z 283.002,A 0.000,B 0.000,C 90.000,E1 36.297} C_DIS
LIN {X -0.127,Y -534.672,Z 282.995,A 0.000,B 0.000,C 90.000,E1 35.152} C_DIS
LIN {X -0.016,Y -533.020,Z 282.986,A 0.000,B 0.000,C 90.000,E1 33.420} C_DIS
LIN {X 0.215,Y -531.171,Z 282.976,A 0.000,B 0.000,C 90.000,E1 31.671} C_DIS
LIN {X -0.016,Y -529.582,Z 282.968,A 0.000,B 0.000,C 90.000,E1 30.256} C_DIS
LIN {X -0.133,Y -527.670,Z 282.958,A 0.000,B 0.000,C 90.000,E1 28.537} C_DIS
LIN {X -0.014,Y -526.068,Z 282.950,A 0.000,B 0.000,C 90.000,E1 27.078} C_DIS
LIN {X 0.166,Y -523.821,Z 282.939,A 0.000,B 0.000,C 90.000,E1 25.027} C_DIS
LIN {X -0.310,Y -522.086,Z 282.930,A 0.000,B 0.000,C 90.000,E1 23.334} C_DIS
LIN {X 0.136,Y -520.427,Z 282.920,A 0.000,B 0.000,C 90.000,E1 21.535} C_DIS
LIN {X 0.006,Y -518.691,Z 282.908,A 0.000,B 0.000,C 90.000,E1 19.504} C_DIS
LIN {X -0.029,Y -517.189,Z 282.897,A 0.000,B 0.000,C 90.000,E1 17.457} C_DIS
LIN {X -0.271,Y -515.643,Z 282.884,A 0.000,B 0.000,C 90.000,E1 15.134} C_DIS
LIN {X -0.121,Y -514.900,Z 282.876,A 0.000,B 0.000,C 90.000,E1 13.647} C_DIS
LIN {X -0.139,Y -514.142,Z 282.866,A 0.000,B 0.000,C 90.000,E1 11.883} C_DIS
LIN {X 0.082,Y -513.435,Z 282.853,A 0.000,B 0.000,C 90.000,E1 9.500} C_DIS
LIN {X 0.216,Y -513.103,Z 282.840,A 0.000,B 0.000,C 90.000,E1 7.125} C_DIS
LIN {X 0.095,Y -513.342,Z 282.823,A 0.000,B 0.000,C 90.000,E1 4.188} C_DIS
LIN {X -0.022,Y -514.083,Z 282.809,A 0.000,B 0.000,C 90.000,E1 1.547} C_DIS
LIN {X -0.018,Y -515.467,Z 282.794,A 0.000,B 0.000,C 90.000,E1 358.912} C_DIS
LIN {X -0.080,Y -517.529,Z 282.779,A 0.000,B 0.000,C 90.000,E1 356.274} C_DIS
LIN {X 0.087,Y -519.548,Z 282.768,A 0.000,B 0.000,C 90.000,E1 354.204} C_DIS
LIN {X -0.227,Y -523.720,Z 282.750,A 0.000,B 0.000,C 90.000,E1 351.027} C_DIS
LIN {X -0.169,Y -528.604,Z 282.736,A 0.000,B 0.000,C 90.000,E1 348.409} C_DIS
LIN {X -0.114,Y -534.884,Z 282.721,A 0.000,B 0.000,C 90.000,E1 345.811} C_DIS
LIN {X 0.087,Y -540.664,Z 282.708,A 0.000,B 0.000,C 90.000,E1 343.504} C_DIS
LIN {X 0.042,Y -548.648,Z 282.693,A 0.000,B 0.000,C 90.000,E1 340.678} C_DIS
LIN {X 0.043,Y -556.689,Z 282.679,A 0.000,B 0.000,C 90.000,E1 338.156} C_DIS
LIN {X -0.012,Y -560.448,Z 282.673,A 0.000,B 0.000,C 90.000,E1 337.050} C_DIS
LIN {X 0.147,Y -567.133,Z 282.662,A 0.000,B 0.000,C 90.000,E1 335.101} C_DIS
LIN {X 0.051,Y -575.038,Z 282.650,A 0.000,B 0.000,C 90.000,E1 332.922} C_DIS
LIN {X 0.078,Y -579.919,Z 282.642,A 0.000,B 0.000,C 90.000,E1 331.563} C_DIS
LIN {X -0.343,Y -582.727,Z 282.638,A 0.000,B 0.000,C 90.000,E1 330.795} C_DIS
LIN {X -0.037,Y -588.207,Z 282.629,A 0.000,B 0.000,C 90.000,E1 329.154} C_DIS
LIN {X -0.111,Y -594.557,Z 282.618,A 0.000,B 0.000,C 90.000,E1 327.296} C_DIS
LIN {X -0.104,Y -602.257,Z 282.607,A 0.000,B 0.000,C 90.000,E1 325.182} C_DIS
LIN {X -0.021,Y -607.126,Z 282.599,A 0.000,B 0.000,C 90.000,E1 323.863} C_DIS
LIN {X -0.270,Y -610.903,Z 282.593,A 0.000,B 0.000,C 90.000,E1 322.844} C_DIS
LIN {X -0.167,Y -615.316,Z 282.586,A 0.000,B 0.000,C 90.000,E1 321.537} C_DIS
LIN {X 0.006,Y -619.532,Z 282.579,A 0.000,B 0.000,C 90.000,E1 320.231} C_DIS
LIN {X 0.002,Y -621.939,Z 282.575,A 0.000,B 0.000,C 90.000,E1 319.461} C_DIS
LIN {X 0.213,Y -625.886,Z 282.568,A 0.000,B 0.000,C 90.000,E1 318.162} C_DIS
LIN {X 0.152,Y -628.809,Z 282.562,A 0.000,B 0.000,C 90.000,E1 317.148} C_DIS
LIN {X -0.095,Y -633.225,Z 282.554,A 0.000,B 0.000,C 90.000,E1 315.648} C_DIS
LIN {X 0.186,Y -637.508,Z 282.545,A 0.000,B 0.000,C 90.000,E1 314.109} C_DIS
LIN {X -0.185,Y -640.249,Z 282.540,A 0.000,B 0.000,C 90.000,E1 313.137} C_DIS
LIN {X -0.060,Y -642.878,Z 282.534,A 0.000,B 0.000,C 90.000,E1 312.123} C_DIS
LIN {X -0.327,Y -645.294,Z 282.529,A 0.000,B 0.000,C 90.000,E1 311.148} C_DIS
LIN {X -0.066,Y -646.928,Z 282.524,A 0.000,B 0.000,C 90.000,E1 310.378} C_DIS
LIN {X 0.222,Y -648.909,Z 282.519,A 0.000,B 0.000,C 90.000,E1 309.358} C_DIS
LIN {X 0.035,Y -650.646,Z 282.513,A 0.000,B 0.000,C 90.000,E1 308.382} C_DIS
LIN {X -0.019,Y -652.236,Z 282.508,A 0.000,B 0.000,C 90.000,E1 307.397} C_DIS
LIN {X -0.179,Y -653.551,Z 282.502,A 0.000,B 0.000,C 90.000,E1 306.423} C_DIS
LIN {X -0.189,Y -654.124,Z 282.500,A 0.000,B 0.000,C 90.000,E1 305.931} C_DIS
LIN {X -0.118,Y -654.593,Z 282.495,A 0.000,B 0.000,C 90.000,E1 305.185} C_DIS
LIN {X -0.115,Y -654.879,Z 282.490,A 0.000,B 0.000,C 90.000,E1 304.199} C_DIS
LIN {X -0.117,Y -655.017,Z 282.485,A 0.000,B 0.000,C 90.000,E1 303.214} C_DIS
LIN {X -0.027,Y -654.724,Z 282.480,A 0.000,B 0.000,C 90.000,E1 302.467} C_DIS
LIN {X -0.385,Y -654.412,Z 282.478,A 0.000,B 0.000,C 90.000,E1 302.005} C_DIS
LIN {X -0.199,Y -653.313,Z 282.472,A 0.000,B 0.000,C 90.000,E1 301.003} C_DIS
LIN {X -0.127,Y -652.121,Z 282.468,A 0.000,B 0.000,C 90.000,E1 300.256} C_DIS
LIN {X -0.299,Y -650.099,Z 282.463,A 0.000,B 0.000,C 90.000,E1 299.283} C_DIS
LIN {X -0.182,Y -647.796,Z 282.457,A 0.000,B 0.000,C 90.000,E1 298.281} C_DIS
LIN {X 0.164,Y -645.322,Z 282.452,A 0.000,B 0.000,C 90.000,E1 297.257} C_DIS
LIN {X -0.025,Y -642.176,Z 282.445,A 0.000,B 0.000,C 90.000,E1 296.027} C_DIS
LIN {X 0.143,Y -637.471,Z 282.435,A 0.000,B 0.000,C 90.000,E1 294.259} C_DIS
LIN {X -0.056,Y -632.781,Z 282.425,A 0.000,B 0.000,C 90.000,E1 292.514} C_DIS
LIN {X -0.009,Y -628.181,Z 282.415,A 0.000,B 0.000,C 90.000,E1 290.737} C_DIS
LIN {X -0.070,Y -623.741,Z 282.405,A 0.000,B 0.000,C 90.000,E1 288.960} C_DIS
LIN {X -0.086,Y -618.959,Z 282.394,A 0.000,B 0.000,C 90.000,E1 286.913} C_DIS
LIN {X 0.301,Y -613.753,Z 282.380,A 0.000,B 0.000,C 90.000,E1 284.300} C_DIS
LIN {X -0.283,Y -608.693,Z 282.362,A 0.000,B 0.000,C 90.000,E1 281.243} C_DIS
LIN {X 0.109,Y -605.685,Z 282.349,A 0.000,B 0.000,C 90.000,E1 278.859} C_DIS
LIN {X -0.044,Y -603.282,Z 282.335,A 0.000,B 0.000,C 90.000,E1 276.258} C_DIS
LIN {X -0.156,Y -601.642,Z 282.319,A 0.000,B 0.000,C 90.000,E1 273.383} C_DIS
LIN {X 0.212,Y -601.143,Z 282.303,A 0.000,B 0.000,C 90.000,E1 270.458} C_DIS
LIN {X -0.207,Y -601.388,Z 282.291,A 0.000,B 0.000,C 90.000,E1 268.396} C_DIS
LIN {X 0.197,Y -602.834,Z 282.275,A 0.000,B 0.000,C 90.000,E1 265.469} C_DIS
LIN {X -0.280,Y -603.876,Z 282.268,A 0.000,B 0.000,C 90.000,E1 264.204} C_DIS
LIN {X -0.158,Y -606.318,Z 282.255,A 0.000,B 0.000,C 90.000,E1 261.837} C_DIS
LIN {X 0.307,Y -610.124,Z 282.239,A 0.000,B 0.000,C 90.000,E1 258.926} C_DIS
LIN {X -0.026,Y -613.378,Z 282.227,A 0.000,B 0.000,C 90.000,E1 256.881} C_DIS
LIN {X 0.234,Y -616.176,Z 282.217,A 0.000,B 0.000,C 90.000,E1 255.046} C_DIS
LIN {X 0.124,Y -617.306,Z 282.213,A 0.000,B 0.000,C 90.000,E1 254.283} C_DIS
LIN {X 0.190,Y -618.225,Z 282.208,A 0.000,B 0.000,C 90.000,E1 253.504} C_DIS
LIN {X 0.269,Y -618.929,Z 282.204,A 0.000,B 0.000,C 90.000,E1 252.725} C_DIS
LIN {X 0.085,Y -619.768,Z 282.197,A 0.000,B 0.000,C 90.000,E1 251.456} C_DIS
LIN {X 0.147,Y -620.239,Z 282.191,A 0.000,B 0.000,C 90.000,E1 250.423} C_DIS
LIN {X -0.347,Y -620.343,Z 282.187,A 0.000,B 0.000,C 90.000,E1 249.699} C_DIS
LIN {X -0.043,Y -620.165,Z 282.183,A 0.000,B 0.000,C 90.000,E1 248.901} C_DIS
LIN {X 0.257,Y -619.791,Z 282.179,A 0.000,B 0.000,C 90.000,E1 248.103} C_DIS
LIN {X -0.021,Y -619.226,Z 282.174,A 0.000,B 0.000,C 90.000,E1 247.358} C_DIS
LIN {X 0.246,Y -617.988,Z 282.169,A 0.000,B 0.000,C 90.000,E1 246.305} C_DIS
LIN {X 0.216,Y -617.283,Z 282.166,A 0.000,B 0.000,C 90.000,E1 245.793} C_DIS
LIN {X -0.092,Y -615.928,Z 282.161,A 0.000,B 0.000,C 90.000,E1 245.049} C_DIS
LIN {X -0.132,Y -614.937,Z 282.159,A 0.000,B 0.000,C 90.000,E1 244.537} C_DIS
LIN {X -0.256,Y -612.010,Z 282.151,A 0.000,B 0.000,C 90.000,E1 243.256} C_DIS
LIN {X -0.391,Y -609.449,Z 282.146,A 0.000,B 0.000,C 90.000,E1 242.231} C_DIS
LIN {X -0.324,Y -606.017,Z 282.138,A 0.000,B 0.000,C 90.000,E1 240.923} C_DIS
LIN {X -0.255,Y -603.163,Z 282.133,A 0.000,B 0.000,C 90.000,E1 239.871} C_DIS
LIN {X 0.002,Y -599.404,Z 282.125,A 0.000,B 0.000,C 90.000,E1 238.535} C_DIS
LIN {X -0.316,Y -595.479,Z 282.118,A 0.000,B 0.000,C 90.000,E1 237.248} C_DIS
LIN {X 0.121,Y -591.414,Z 282.111,A 0.000,B 0.000,C 90.000,E1 235.881} C_DIS
LIN {X -0.011,Y -587.075,Z 282.103,A 0.000,B 0.000,C 90.000,E1 234.562} C_DIS
LIN {X -0.280,Y -578.612,Z 282.088,A 0.000,B 0.000,C 90.000,E1 231.904} C_DIS
LIN {X -0.092,Y -575.231,Z 282.082,A 0.000,B 0.000,C 90.000,E1 230.803} C_DIS
LIN {X -0.258,Y -570.976,Z 282.075,A 0.000,B 0.000,C 90.000,E1 229.461} C_DIS
LIN {X -0.125,Y -566.775,Z 282.067,A 0.000,B 0.000,C 90.000,E1 228.081} C_DIS
LIN {X -0.005,Y -561.659,Z 282.058,A 0.000,B 0.000,C 90.000,E1 226.419} C_DIS
LIN {X 0.057,Y -555.602,Z 282.047,A 0.000,B 0.000,C 90.000,E1 224.474} C_DIS
LIN {X -0.144,Y -552.169,Z 282.041,A 0.000,B 0.000,C 90.000,E1 223.380} C_DIS
LIN {X 0.061,Y -546.963,Z 282.032,A 0.000,B 0.000,C 90.000,E1 221.676} C_DIS
LIN {X 0.181,Y -542.633,Z 282.024,A 0.000,B 0.000,C 90.000,E1 220.253} C_DIS
LIN {X 0.223,Y -538.273,Z 282.016,A 0.000,B 0.000,C 90.000,E1 218.830} C_DIS
LIN {X -0.153,Y -532.241,Z 282.005,A 0.000,B 0.000,C 90.000,E1 216.870} C_DIS
LIN {X 0.168,Y -526.284,Z 281.994,A 0.000,B 0.000,C 90.000,E1 214.818} C_DIS
LIN {X 0.030,Y -520.561,Z 281.982,A 0.000,B 0.000,C 90.000,E1 212.801} C_DIS
LIN {X 0.067,Y -515.091,Z 281.971,A 0.000,B 0.000,C 90.000,E1 210.747} C_DIS
LIN {X -0.044,Y -508.319,Z 281.956,A 0.000,B 0.000,C 90.000,E1 208.103} C_DIS
LIN {X -0.036,Y -502.761,Z 281.943,A 0.000,B 0.000,C 90.000,E1 205.720} C_DIS
LIN {X 0.157,Y -498.913,Z 281.933,A 0.000,B 0.000,C 90.000,E1 203.898} C_DIS
LIN {X 0.014,Y -495.778,Z 281.925,A 0.000,B 0.000,C 90.000,E1 202.408} C_DIS
LIN {X -0.187,Y -492.796,Z 281.916,A 0.000,B 0.000,C 90.000,E1 200.918} C_DIS
LIN {X -0.130,Y -489.476,Z 281.906,A 0.000,B 0.000,C 90.000,E1 199.087} C_DIS
LIN {X 0.032,Y -485.383,Z 281.892,A 0.000,B 0.000,C 90.000,E1 196.622} C_DIS
LIN {X 0.109,Y -480.759,Z 281.875,A 0.000,B 0.000,C 90.000,E1 193.536} C_DIS
LIN {X -0.161,Y -477.073,Z 281.860,A 0.000,B 0.000,C 90.000,E1 190.782} C_DIS
LIN {X -0.258,Y -473.845,Z 281.844,A 0.000,B 0.000,C 90.000,E1 187.992} C_DIS
LIN {X -0.185,Y -471.569,Z 281.832,A 0.000,B 0.000,C 90.000,E1 185.796} C_DIS
LIN {X 0.197,Y -469.597,Z 281.820,A 0.000,B 0.000,C 90.000,E1 183.555} C_DIS
LIN {X 0.026,Y -467.882,Z 281.808,A 0.000,B 0.000,C 90.000,E1 181.375} C_DIS
LIN {X -0.212,Y -466.475,Z 281.795,A 0.000,B 0.000,C 90.000,E1 179.198} C_DIS
LIN {X 0.232,Y -465.280,Z 281.781,A 0.000,B 0.000,C 90.000,E1 176.617} C_DIS
LIN {X 0.193,Y -464.334,Z 281.764,A 0.000,B 0.000,C 90.000,E1 173.457} C_DIS
LIN {X -0.172,Y -464.101,Z 281.753,A 0.000,B 0.000,C 90.000,E1 171.602} C_DIS
LIN {X 0.178,Y -463.968,Z 281.741,A 0.000,B 0.000,C 90.000,E1 169.342} C_DIS
LIN {X -0.217,Y -464.170,Z 281.729,A 0.000,B 0.000,C 90.000,E1 167.173} C_DIS
LIN {X -0.009,Y -464.468,Z 281.722,A 0.000,B 0.000,C 90.000,E1 165.880} C_DIS
LIN {X 0.089,Y -466.076,Z 281.701,A 0.000,B 0.000,C 90.000,E1 162.072} C_DIS
LIN {X -0.051,Y -467.566,Z 281.688,A 0.000,B 0.000,C 90.000,E1 159.880} C_DIS
LIN {X -0.026,Y -469.676,Z 281.674,A 0.000,B 0.000,C 90.000,E1 157.358} C_DIS
LIN {X 0.002,Y -472.312,Z 281.660,A 0.000,B 0.000,C 90.000,E1 154.845} C_DIS
LIN {X -0.016,Y -477.190,Z 281.639,A 0.000,B 0.000,C 90.000,E1 151.101} C_DIS
LIN {X -0.127,Y -480.095,Z 281.629,A 0.000,B 0.000,C 90.000,E1 149.253} C_DIS
LIN {X 0.102,Y -484.113,Z 281.615,A 0.000,B 0.000,C 90.000,E1 146.755} C_DIS
LIN {X 0.244,Y -487.254,Z 281.605,A 0.000,B 0.000,C 90.000,E1 144.895} C_DIS
LIN {X 0.042,Y -490.414,Z 281.595,A 0.000,B 0.000,C 90.000,E1 143.084} C_DIS
LIN {X -0.285,Y -492.469,Z 281.588,A 0.000,B 0.000,C 90.000,E1 141.904} C_DIS
LIN {X -0.174,Y -495.323,Z 281.578,A 0.000,B 0.000,C 90.000,E1 140.070} C_DIS
LIN {X 0.080,Y -497.368,Z 281.570,A 0.000,B 0.000,C 90.000,E1 138.528} C_DIS
LIN {X -0.014,Y -498.440,Z 281.565,A 0.000,B 0.000,C 90.000,E1 137.634} C_DIS
LIN {X -0.128,Y -499.227,Z 281.560,A 0.000,B 0.000,C 90.000,E1 136.743} C_DIS
LIN {X -0.013,Y -499.889,Z 281.553,A 0.000,B 0.000,C 90.000,E1 135.526} C_DIS
LIN {X 0.246,Y -500.166,Z 281.548,A 0.000,B 0.000,C 90.000,E1 134.595} C_DIS
LIN {X 0.155,Y -500.132,Z 281.543,A 0.000,B 0.000,C 90.000,E1 133.704} C_DIS
LIN {X -0.143,Y -500.044,Z 281.540,A 0.000,B 0.000,C 90.000,E1 133.137} C_DIS
LIN {X 0.125,Y -499.614,Z 281.535,A 0.000,B 0.000,C 90.000,E1 132.204} C_DIS
LIN {X 0.055,Y -498.936,Z 281.530,A 0.000,B 0.000,C 90.000,E1 131.310} C_DIS
LIN {X 0.176,Y -497.688,Z 281.523,A 0.000,B 0.000,C 90.000,E1 130.092} C_DIS
LIN {X 0.090,Y -496.594,Z 281.518,A 0.000,B 0.000,C 90.000,E1 129.197} C_DIS
LIN {X 0.104,Y -494.595,Z 281.509,A 0.000,B 0.000,C 90.000,E1 127.684} C_DIS
LIN {X -0.020,Y -493.266,Z 281.504,A 0.000,B 0.000,C 90.000,E1 126.790} C_DIS
LIN {X -0.212,Y -491.281,Z 281.498,A 0.000,B 0.000,C 90.000,E1 125.598} C_DIS
LIN {X 0.088,Y -488.564,Z 281.489,A 0.000,B 0.000,C 90.000,E1 124.040} C_DIS
LIN {X -0.213,Y -485.663,Z 281.481,A 0.000,B 0.000,C 90.000,E1 122.546} C_DIS
LIN {X -0.126,Y -481.648,Z 281.469,A 0.000,B 0.000,C 90.000,E1 120.384} C_DIS
LIN {X 0.032,Y -478.710,Z 281.460,A 0.000,B 0.000,C 90.000,E1 118.821} C_DIS
LIN {X -0.136,Y -474.605,Z 281.448,A 0.000,B 0.000,C 90.000,E1 116.668} C_DIS
LIN {X 0.052,Y -470.985,Z 281.438,A 0.000,B 0.000,C 90.000,E1 114.771} C_DIS
LIN {X 0.020,Y -468.061,Z 281.429,A 0.000,B 0.000,C 90.000,E1 113.206} C_DIS
LIN {X 0.233,Y -464.047,Z 281.417,A 0.000,B 0.000,C 90.000,E1 110.972} C_DIS
LIN {X 0.178,Y -459.936,Z 281.404,A 0.000,B 0.000,C 90.000,E1 108.598} C_DIS
LIN {X 0.012,Y -459.721,Z 281.403,A 0.000,B 0.000,C 90.000,E1 108.489} C_DIS
LIN {X -0.029,Y -459.724,Z 281.403,A 0.000,B 0.000,C 90.000,E1 108.489} C_DIS
LIN {X 0.120,Y -467.604,Z 281.383,A 0.000,B 0.000,C 90.000,E1 104.954} C_DIS
LIN {X -0.148,Y -468.597,Z 281.380,A 0.000,B 0.000,C 90.000,E1 104.356} C_DIS
LIN {X 0.079,Y -475.830,Z 281.357,A 0.000,B 0.000,C 90.000,E1 100.254} C_DIS
LIN {X -0.083,Y -476.318,Z 281.355,A 0.000,B 0.000,C 90.000,E1 99.962} C_DIS
LIN {X -0.136,Y -481.811,Z 281.331,A 0.000,B 0.000,C 90.000,E1 95.625} C_DIS
LIN {X 0.191,Y -482.177,Z 281.329,A 0.000,B 0.000,C 90.000,E1 95.277} C_DIS
LIN {X 0.125,Y -485.322,Z 281.306,A 0.000,B 0.000,C 90.000,E1 90.974} C_DIS
LIN {X -0.050,Y -485.535,Z 281.304,A 0.000,B 0.000,C 90.000,E1 90.688} C_DIS
LIN {X 0.157,Y -486.326,Z 281.282,A 0.000,B 0.000,C 90.000,E1 86.674} C_DIS
LIN {X -0.194,Y -486.295,Z 281.278,A 0.000,B 0.000,C 90.000,E1 86.102} C_DIS
LIN {X 0.011,Y -484.695,Z 281.254,A 0.000,B 0.000,C 90.000,E1 81.781} C_DIS
LIN {X -0.121,Y -484.583,Z 281.253,A 0.000,B 0.000,C 90.000,E1 81.489} C_DIS
LIN {X -0.240,Y -480.520,Z 281.227,A 0.000,B 0.000,C 90.000,E1 76.881} C_DIS
LIN {X 0.124,Y -474.271,Z 281.201,A 0.000,B 0.000,C 90.000,E1 72.181} C_DIS
LIN {X 0.092,Y -473.819,Z 281.199,A 0.000,B 0.000,C 90.000,E1 71.873} C_DIS
LIN {X 0.169,Y -471.812,Z 281.194,A 0.000,B 0.000,C 90.000,E1 70.859} C_DIS
LIN {X 0.128,Y -471.812,Z 281.194,A 0.000,B 0.000,C 90.000,E1 70.859} C_DIS
LIN {X -0.021,Y -474.745,Z 281.187,A 0.000,B 0.000,C 90.000,E1 69.699} C_DIS
LIN {X -0.167,Y -480.361,Z 281.175,A 0.000,B 0.000,C 90.000,E1 67.539} C_DIS
LIN {X 0.022,Y -486.132,Z 281.163,A 0.000,B 0.000,C 90.000,E1 65.357} C_DIS
LIN {X 0.074,Y -490.377,Z 281.155,A 0.000,B 0.000,C 90.000,E1 63.819} C_DIS
LIN {X -0.193,Y -495.493,Z 281.145,A 0.000,B 0.000,C 90.000,E1 62.025} C_DIS
LIN {X -0.124,Y -500.737,Z 281.134,A 0.000,B 0.000,C 90.000,E1 60.205} C_DIS
LIN {X 0.185,Y -506.880,Z 281.123,A 0.000,B 0.000,C 90.000,E1 58.074} C_DIS
LIN {X -0.082,Y -510.367,Z 281.116,A 0.000,B 0.000,C 90.000,E1 56.914} C_DIS
LIN {X -0.092,Y -514.606,Z 281.108,A 0.000,B 0.000,C 90.000,E1 55.435} C_DIS
LIN {X -0.253,Y -517.815,Z 281.101,A 0.000,B 0.000,C 90.000,E1 54.276} C_DIS
LIN {X 0.184,Y -521.519,Z 281.093,A 0.000,B 0.000,C 90.000,E1 52.763} C_DIS
LIN {X -0.001,Y -524.262,Z 281.087,A 0.000,B 0.000,C 90.000,E1 51.618} C_DIS
LIN {X 0.177,Y -526.753,Z 281.080,A 0.000,B 0.000,C 90.000,E1 50.436} C_DIS
LIN {X -0.012,Y -529.044,Z 281.074,A 0.000,B 0.000,C 90.000,E1 49.299} C_DIS
LIN {X -0.168,Y -531.010,Z 281.068,A 0.000,B 0.000,C 90.000,E1 48.162} C_DIS
LIN {X -0.279,Y -532.287,Z 281.063,A 0.000,B 0.000,C 90.000,E1 47.310} C_DIS
LIN {X -0.035,Y -533.744,Z 281.056,A 0.000,B 0.000,C 90.000,E1 46.134} C_DIS
LIN {X -0.153,Y -534.792,Z 281.050,A 0.000,B 0.000,C 90.000,E1 45.000} C_DIS
LIN {X 0.096,Y -535.737,Z 281.042,A 0.000,B 0.000,C 90.000,E1 43.542} C_DIS
LIN {X -0.015,Y -536.272,Z 281.034,A 0.000,B 0.000,C 90.000,E1 42.123} C_DIS
LIN {X -0.074,Y -536.451,Z 281.029,A 0.000,B 0.000,C 90.000,E1 41.272} C_DIS
LIN {X 0.277,Y -536.406,Z 281.023,A 0.000,B 0.000,C 90.000,E1 40.092} C_DIS
LIN {X -0.127,Y -536.213,Z 281.018,A 0.000,B 0.000,C 90.000,E1 39.277} C_DIS
LIN {X 0.227,Y -535.735,Z 281.012,A 0.000,B 0.000,C 90.000,E1 38.096} C_DIS
LIN {X 0.245,Y -534.632,Z 281.002,A 0.000,B 0.000,C 90.000,E1 36.377} C_DIS
LIN {X 0.241,Y -533.667,Z 280.996,A 0.000,B 0.000,C 90.000,E1 35.231} C_DIS
LIN {X 0.332,Y -532.004,Z 280.986,A 0.000,B 0.000,C 90.000,E1 33.499} C_DIS
LIN {X 0.093,Y -530.119,Z 280.977,A 0.000,B 0.000,C 90.000,E1 31.799} C_DIS
LIN {X -0.157,Y -528.522,Z 280.969,A 0.000,B 0.000,C 90.000,E1 30.384} C_DIS
LIN {X -0.144,Y -526.241,Z 280.958,A 0.000,B 0.000,C 90.000,E1 28.359} C_DIS
LIN {X -0.117,Y -524.285,Z 280.948,A 0.000,B 0.000,C 90.000,E1 26.616} C_DIS
LIN {X 0.158,Y -521.769,Z 280.935,A 0.000,B 0.000,C 90.000,E1 24.259} C_DIS
LIN {X 0.288,Y -520.603,Z 280.928,A 0.000,B 0.000,C 90.000,E1 23.078} C_DIS
LIN {X -0.125,Y -519.239,Z 280.920,A 0.000,B 0.000,C 90.000,E1 21.663} C_DIS
LIN {X 0.208,Y -517.449,Z 280.909,A 0.000,B 0.000,C 90.000,E1 19.577} C_DIS
LIN {X 0.152,Y -515.910,Z 280.898,A 0.000,B 0.000,C 90.000,E1 17.528} C_DIS
LIN {X 0.049,Y -514.496,Z 280.886,A 0.000,B 0.000,C 90.000,E1 15.481} C_DIS
LIN {X 0.022,Y -513.564,Z 280.876,A 0.000,B 0.000,C 90.000,E1 13.716} C_DIS
LIN {X -0.042,Y -512.666,Z 280.865,A 0.000,B 0.000,C 90.000,E1 11.658} C_DIS
LIN {X -0.240,Y -512.037,Z 280.853,A 0.000,B 0.000,C 90.000,E1 9.613} C_DIS
LIN {X -0.193,Y -511.639,Z 280.839,A 0.000,B 0.000,C 90.000,E1 6.947} C_DIS
LIN {X 0.176,Y -511.806,Z 280.824,A 0.000,B 0.000,C 90.000,E1 4.245} C_DIS
LIN {X 0.007,Y -512.533,Z 280.809,A 0.000,B 0.000,C 90.000,E1 1.604} C_DIS
LIN {X -0.035,Y -513.872,Z 280.794,A 0.000,B 0.000,C 90.000,E1 358.912} C_DIS
LIN {X -0.149,Y -515.936,Z 280.779,A 0.000,B 0.000,C 90.000,E1 356.274} C_DIS
LIN {X -0.025,Y -517.989,Z 280.768,A 0.000,B 0.000,C 90.000,E1 354.204} C_DIS
LIN {X 0.192,Y -521.669,Z 280.752,A 0.000,B 0.000,C 90.000,E1 351.254} C_DIS
LIN {X 0.224,Y -527.054,Z 280.735,A 0.000,B 0.000,C 90.000,E1 348.342} C_DIS
LIN {X 0.119,Y -533.346,Z 280.721,A 0.000,B 0.000,C 90.000,E1 345.755} C_DIS
LIN {X 0.219,Y -538.398,Z 280.710,A 0.000,B 0.000,C 90.000,E1 343.740} C_DIS
LIN {X 0.074,Y -543.837,Z 280.699,A 0.000,B 0.000,C 90.000,E1 341.764} C_DIS
LIN {X 0.240,Y -551.619,Z 280.685,A 0.000,B 0.000,C 90.000,E1 339.209} C_DIS
LIN {X 0.037,Y -559.062,Z 280.672,A 0.000,B 0.000,C 90.000,E1 336.997} C_DIS
LIN {X 0.154,Y -565.808,Z 280.662,A 0.000,B 0.000,C 90.000,E1 335.049} C_DIS
LIN {X 0.011,Y -573.724,Z 280.649,A 0.000,B 0.000,C 90.000,E1 332.871} C_DIS
LIN {X 0.009,Y -578.654,Z 280.642,A 0.000,B 0.000,C 90.000,E1 331.513} C_DIS
LIN {X -0.146,Y -581.473,Z 280.637,A 0.000,B 0.000,C 90.000,E1 330.717} C_DIS
LIN {X 0.141,Y -586.972,Z 280.628,A 0.000,B 0.000,C 90.000,E1 329.076} C_DIS
LIN {X -0.178,Y -595.227,Z 280.615,A 0.000,B 0.000,C 90.000,E1 326.707} C_DIS
LIN {X 0.027,Y -601.066,Z 280.606,A 0.000,B 0.000,C 90.000,E1 325.102} C_DIS
LIN {X 0.093,Y -605.959,Z 280.599,A 0.000,B 0.000,C 90.000,E1 323.783} C_DIS
LIN {X -0.167,Y -609.751,Z 280.593,A 0.000,B 0.000,C 90.000,E1 322.763} C_DIS
LIN {X -0.081,Y -614.182,Z 280.586,A 0.000,B 0.000,C 90.000,E1 321.457} C_DIS
LIN {X 0.075,Y -618.416,Z 280.579,A 0.000,B 0.000,C 90.000,E1 320.150} C_DIS
LIN {X 0.060,Y -620.811,Z 280.574,A 0.000,B 0.000,C 90.000,E1 319.380} C_DIS
LIN {X 0.254,Y -624.801,Z 280.567,A 0.000,B 0.000,C 90.000,E1 318.081} C_DIS
LIN {X 0.180,Y -627.750,Z 280.562,A 0.000,B 0.000,C 90.000,E1 317.067} C_DIS
LIN {X -0.087,Y -632.167,Z 280.553,A 0.000,B 0.000,C 90.000,E1 315.567} C_DIS
LIN {X 0.172,Y -636.462,Z 280.545,A 0.000,B 0.000,C 90.000,E1 314.028} C_DIS
LIN {X 0.072,Y -640.524,Z 280.536,A 0.000,B 0.000,C 90.000,E1 312.528} C_DIS
LIN {X 0.204,Y -643.006,Z 280.531,A 0.000,B 0.000,C 90.000,E1 311.515} C_DIS
LIN {X -0.058,Y -645.291,Z 280.525,A 0.000,B 0.000,C 90.000,E1 310.539} C_DIS
LIN {X 0.133,Y -647.703,Z 280.518,A 0.000,B 0.000,C 90.000,E1 309.277} C_DIS
LIN {X -0.072,Y -649.405,Z 280.513,A 0.000,B 0.000,C 90.000,E1 308.302} C_DIS
LIN {X -0.145,Y -650.936,Z 280.507,A 0.000,B 0.000,C 90.000,E1 307.317} C_DIS
LIN {X -0.245,Y -651.932,Z 280.503,A 0.000,B 0.000,C 90.000,E1 306.583} C_DIS
LIN {X -0.263,Y -652.515,Z 280.500,A 0.000,B 0.000,C 90.000,E1 306.091} C_DIS
LIN {X 0.173,Y -653.058,Z 280.496,A 0.000,B 0.000,C 90.000,E1 305.311} C_DIS
LIN {X 0.153,Y -653.371,Z 280.491,A 0.000,B 0.000,C 90.000,E1 304.326} C_DIS
LIN {X -0.232,Y -653.538,Z 280.485,A 0.000,B 0.000,C 90.000,E1 303.372} C_DIS
LIN {X -0.152,Y -653.319,Z 280.481,A 0.000,B 0.000,C 90.000,E1 302.625} C_DIS
LIN {X -0.073,Y -652.804,Z 280.477,A 0.000,B 0.000,C 90.000,E1 301.878} C_DIS
LIN {X 0.093,Y -651.685,Z 280.472,A 0.000,B 0.000,C 90.000,E1 300.875} C_DIS
LIN {X 0.149,Y -650.444,Z 280.467,A 0.000,B 0.000,C 90.000,E1 300.129} C_DIS
LIN {X 0.048,Y -647.820,Z 280.461,A 0.000,B 0.000,C 90.000,E1 298.899} C_DIS
LIN {X 0.133,Y -645.483,Z 280.455,A 0.000,B 0.000,C 90.000,E1 297.897} C_DIS
LIN {X 0.018,Y -641.688,Z 280.447,A 0.000,B 0.000,C 90.000,E1 296.411} C_DIS
LIN {X 0.003,Y -639.026,Z 280.441,A 0.000,B 0.000,C 90.000,E1 295.412} C_DIS
LIN {X 0.108,Y -634.336,Z 280.431,A 0.000,B 0.000,C 90.000,E1 293.643} C_DIS
LIN {X -0.157,Y -629.659,Z 280.422,A 0.000,B 0.000,C 90.000,E1 291.897} C_DIS
LIN {X 0.036,Y -625.792,Z 280.413,A 0.000,B 0.000,C 90.000,E1 290.355} C_DIS
LIN {X 0.293,Y -621.366,Z 280.403,A 0.000,B 0.000,C 90.000,E1 288.544} C_DIS
LIN {X -0.093,Y -617.810,Z 280.395,A 0.000,B 0.000,C 90.000,E1 287.040} C_DIS
LIN {X 0.024,Y -612.100,Z 280.379,A 0.000,B 0.000,C 90.000,E1 284.189} C_DIS
LIN {X -0.011,Y -607.099,Z 280.362,A 0.000,B 0.000,C 90.000,E1 281.074} C_DIS
LIN {X -0.204,Y -604.749,Z 280.351,A 0.000,B 0.000,C 90.000,E1 279.265} C_DIS
LIN {X 0.210,Y -602.228,Z 280.337,A 0.000,B 0.000,C 90.000,E1 276.606} C_DIS
LIN {X 0.107,Y -600.448,Z 280.321,A 0.000,B 0.000,C 90.000,E1 273.726} C_DIS
LIN {X 0.063,Y -599.791,Z 280.303,A 0.000,B 0.000,C 90.000,E1 270.573} C_DIS
LIN {X 0.208,Y -600.026,Z 280.292,A 0.000,B 0.000,C 90.000,E1 268.453} C_DIS
LIN {X -0.279,Y -601.262,Z 280.277,A 0.000,B 0.000,C 90.000,E1 265.869} C_DIS
LIN {X -0.175,Y -602.276,Z 280.270,A 0.000,B 0.000,C 90.000,E1 264.546} C_DIS
LIN {X 0.146,Y -604.917,Z 280.255,A 0.000,B 0.000,C 90.000,E1 261.894} C_DIS
LIN {X -0.150,Y -608.713,Z 280.239,A 0.000,B 0.000,C 90.000,E1 259.050} C_DIS
LIN {X 0.199,Y -611.968,Z 280.228,A 0.000,B 0.000,C 90.000,E1 256.937} C_DIS
LIN {X 0.163,Y -613.969,Z 280.220,A 0.000,B 0.000,C 90.000,E1 255.644} C_DIS
LIN {X -0.046,Y -615.592,Z 280.215,A 0.000,B 0.000,C 90.000,E1 254.629} C_DIS
LIN {X -0.227,Y -616.898,Z 280.209,A 0.000,B 0.000,C 90.000,E1 253.614} C_DIS
LIN {X -0.158,Y -617.637,Z 280.205,A 0.000,B 0.000,C 90.000,E1 252.834} C_DIS
LIN {X 0.035,Y -618.467,Z 280.197,A 0.000,B 0.000,C 90.000,E1 251.529} C_DIS
LIN {X 0.311,Y -618.860,Z 280.193,A 0.000,B 0.000,C 90.000,E1 250.732} C_DIS
LIN {X -0.222,Y -619.093,Z 280.187,A 0.000,B 0.000,C 90.000,E1 249.752} C_DIS
LIN {X -0.175,Y -618.852,Z 280.182,A 0.000,B 0.000,C 90.000,E1 248.720} C_DIS
LIN {X 0.110,Y -618.412,Z 280.177,A 0.000,B 0.000,C 90.000,E1 247.922} C_DIS
LIN {X -0.183,Y -617.767,Z 280.173,A 0.000,B 0.000,C 90.000,E1 247.177} C_DIS
LIN {X 0.311,Y -616.449,Z 280.167,A 0.000,B 0.000,C 90.000,E1 246.102} C_DIS
LIN {X 0.019,Y -615.658,Z 280.165,A 0.000,B 0.000,C 90.000,E1 245.613} C_DIS
LIN {X -0.070,Y -613.766,Z 280.159,A 0.000,B 0.000,C 90.000,E1 244.588} C_DIS
LIN {X -0.177,Y -611.449,Z 280.153,A 0.000,B 0.000,C 90.000,E1 243.563} C_DIS
LIN {X 0.228,Y -608.952,Z 280.147,A 0.000,B 0.000,C 90.000,E1 242.487} C_DIS
LIN {X 0.283,Y -605.550,Z 280.140,A 0.000,B 0.000,C 90.000,E1 241.179} C_DIS
LIN {X 0.280,Y -602.041,Z 280.133,A 0.000,B 0.000,C 90.000,E1 239.871} C_DIS
LIN {X 0.003,Y -598.280,Z 280.126,A 0.000,B 0.000,C 90.000,E1 238.584} C_DIS
LIN {X 0.175,Y -594.351,Z 280.118,A 0.000,B 0.000,C 90.000,E1 237.248} C_DIS
LIN {X 0.098,Y -590.260,Z 280.111,A 0.000,B 0.000,C 90.000,E1 235.928} C_DIS
LIN {X -0.045,Y -585.916,Z 280.103,A 0.000,B 0.000,C 90.000,E1 234.609} C_DIS
LIN {X -0.046,Y -578.284,Z 280.090,A 0.000,B 0.000,C 90.000,E1 232.190} C_DIS
LIN {X 0.287,Y -574.077,Z 280.082,A 0.000,B 0.000,C 90.000,E1 230.803} C_DIS
LIN {X 0.099,Y -569.846,Z 280.075,A 0.000,B 0.000,C 90.000,E1 229.461} C_DIS
LIN {X -0.105,Y -564.766,Z 280.066,A 0.000,B 0.000,C 90.000,E1 227.838} C_DIS
LIN {X -0.024,Y -559.630,Z 280.057,A 0.000,B 0.000,C 90.000,E1 226.176} C_DIS
LIN {X -0.014,Y -553.571,Z 280.046,A 0.000,B 0.000,C 90.000,E1 224.231} C_DIS
LIN {X 0.158,Y -550.070,Z 280.040,A 0.000,B 0.000,C 90.000,E1 223.095} C_DIS
LIN {X -0.086,Y -544.869,Z 280.030,A 0.000,B 0.000,C 90.000,E1 221.434} C_DIS
LIN {X -0.006,Y -540.531,Z 280.022,A 0.000,B 0.000,C 90.000,E1 220.011} C_DIS
LIN {X 0.000,Y -535.268,Z 280.013,A 0.000,B 0.000,C 90.000,E1 218.302} C_DIS
LIN {X -0.006,Y -530.996,Z 280.005,A 0.000,B 0.000,C 90.000,E1 216.870} C_DIS
LIN {X 0.282,Y -525.034,Z 279.994,A 0.000,B 0.000,C 90.000,E1 214.818} C_DIS
LIN {X 0.167,Y -520.118,Z 279.984,A 0.000,B 0.000,C 90.000,E1 213.086} C_DIS
LIN {X 0.115,Y -513.833,Z 279.971,A 0.000,B 0.000,C 90.000,E1 210.747} C_DIS
LIN {X -0.121,Y -507.778,Z 279.958,A 0.000,B 0.000,C 90.000,E1 208.409} C_DIS
LIN {X 0.015,Y -502.865,Z 279.946,A 0.000,B 0.000,C 90.000,E1 206.309} C_DIS
LIN {X 0.098,Y -497.651,Z 279.933,A 0.000,B 0.000,C 90.000,E1 203.898} C_DIS
LIN {X 0.121,Y -494.540,Z 279.924,A 0.000,B 0.000,C 90.000,E1 202.386} C_DIS
LIN {X -0.182,Y -489.891,Z 279.911,A 0.000,B 0.000,C 90.000,E1 199.993} C_DIS
LIN {X 0.003,Y -484.661,Z 279.894,A 0.000,B 0.000,C 90.000,E1 196.913} C_DIS
LIN {X -0.254,Y -480.808,Z 279.880,A 0.000,B 0.000,C 90.000,E1 194.481} C_DIS
LIN {X 0.182,Y -478.666,Z 279.872,A 0.000,B 0.000,C 90.000,E1 192.883} C_DIS
LIN {X 0.147,Y -475.913,Z 279.860,A 0.000,B 0.000,C 90.000,E1 190.715} C_DIS
LIN {X -0.076,Y -472.688,Z 279.844,A 0.000,B 0.000,C 90.000,E1 187.936} C_DIS
LIN {X -0.033,Y -470.437,Z 279.832,A 0.000,B 0.000,C 90.000,E1 185.739} C_DIS
LIN {X -0.148,Y -468.473,Z 279.820,A 0.000,B 0.000,C 90.000,E1 183.555} C_DIS
LIN {X 0.120,Y -466.787,Z 279.807,A 0.000,B 0.000,C 90.000,E1 181.318} C_DIS
LIN {X -0.148,Y -465.390,Z 279.795,A 0.000,B 0.000,C 90.000,E1 179.141} C_DIS
LIN {X -0.202,Y -464.195,Z 279.781,A 0.000,B 0.000,C 90.000,E1 176.617} C_DIS
LIN {X -0.018,Y -463.369,Z 279.765,A 0.000,B 0.000,C 90.000,E1 173.742} C_DIS
LIN {X -0.209,Y -463.079,Z 279.753,A 0.000,B 0.000,C 90.000,E1 171.546} C_DIS
LIN {X -0.141,Y -462.959,Z 279.742,A 0.000,B 0.000,C 90.000,E1 169.634} C_DIS
LIN {X -0.111,Y -463.176,Z 279.730,A 0.000,B 0.000,C 90.000,E1 167.409} C_DIS
LIN {X -0.011,Y -463.504,Z 279.721,A 0.000,B 0.000,C 90.000,E1 165.811} C_DIS
LIN {X 0.135,Y -464.974,Z 279.702,A 0.000,B 0.000,C 90.000,E1 162.308} C_DIS
LIN {X -0.029,Y -466.448,Z 279.690,A 0.000,B 0.000,C 90.000,E1 160.115} C_DIS
LIN {X -0.027,Y -468.539,Z 279.676,A 0.000,B 0.000,C 90.000,E1 157.592} C_DIS
LIN {X -0.267,Y -471.446,Z 279.660,A 0.000,B 0.000,C 90.000,E1 154.793} C_DIS
LIN {X 0.120,Y -475.905,Z 279.641,A 0.000,B 0.000,C 90.000,E1 151.307} C_DIS
LIN {X -0.023,Y -478.766,Z 279.630,A 0.000,B 0.000,C 90.000,E1 149.459} C_DIS
LIN {X -0.052,Y -482.249,Z 279.618,A 0.000,B 0.000,C 90.000,E1 147.296} C_DIS
LIN {X -0.224,Y -485.378,Z 279.608,A 0.000,B 0.000,C 90.000,E1 145.468} C_DIS
LIN {X -0.180,Y -488.543,Z 279.598,A 0.000,B 0.000,C 90.000,E1 143.623} C_DIS
LIN {X -0.141,Y -490.648,Z 279.591,A 0.000,B 0.000,C 90.000,E1 142.396} C_DIS
LIN {X -0.224,Y -493.060,Z 279.583,A 0.000,B 0.000,C 90.000,E1 140.884} C_DIS
LIN {X -0.044,Y -494.461,Z 279.578,A 0.000,B 0.000,C 90.000,E1 139.952} C_DIS
LIN {X -0.123,Y -496.480,Z 279.569,A 0.000,B 0.000,C 90.000,E1 138.447} C_DIS
LIN {X -0.227,Y -497.532,Z 279.564,A 0.000,B 0.000,C 90.000,E1 137.553} C_DIS
LIN {X 0.012,Y -498.287,Z 279.559,A 0.000,B 0.000,C 90.000,E1 136.620} C_DIS
LIN {X 0.100,Y -498.931,Z 279.552,A 0.000,B 0.000,C 90.000,E1 135.405} C_DIS
LIN {X -0.002,Y -499.201,Z 279.547,A 0.000,B 0.000,C 90.000,E1 134.514} C_DIS
LIN {X 0.097,Y -499.112,Z 279.541,A 0.000,B 0.000,C 90.000,E1 133.299} C_DIS
LIN {X 0.017,Y -498.759,Z 279.536,A 0.000,B 0.000,C 90.000,E1 132.405} C_DIS
LIN {X -0.097,Y -498.172,Z 279.531,A 0.000,B 0.000,C 90.000,E1 131.515} C_DIS
LIN {X -0.180,Y -497.349,Z 279.526,A 0.000,B 0.000,C 90.000,E1 130.620} C_DIS
LIN {X -0.088,Y -495.987,Z 279.519,A 0.000,B 0.000,C 90.000,E1 129.402} C_DIS
LIN {X -0.090,Y -493.993,Z 279.510,A 0.000,B 0.000,C 90.000,E1 127.890} C_DIS
LIN {X 0.172,Y -492.697,Z 279.505,A 0.000,B 0.000,C 90.000,E1 126.950} C_DIS
LIN {X 0.262,Y -490.749,Z 279.499,A 0.000,B 0.000,C 90.000,E1 125.724} C_DIS
LIN {X -0.131,Y -488.060,Z 279.490,A 0.000,B 0.000,C 90.000,E1 124.246} C_DIS
LIN {X 0.000,Y -485.772,Z 279.483,A 0.000,B 0.000,C 90.000,E1 123.007} C_DIS
LIN {X 0.279,Y -482.258,Z 279.473,A 0.000,B 0.000,C 90.000,E1 121.131} C_DIS
LIN {X 0.033,Y -479.442,Z 279.465,A 0.000,B 0.000,C 90.000,E1 119.617} C_DIS
LIN {X -0.263,Y -476.498,Z 279.456,A 0.000,B 0.000,C 90.000,E1 118.103} C_DIS
LIN {X -0.240,Y -472.996,Z 279.446,A 0.000,B 0.000,C 90.000,E1 116.232} C_DIS
LIN {X -0.129,Y -468.808,Z 279.433,A 0.000,B 0.000,C 90.000,E1 114.027} C_DIS
LIN {X 0.117,Y -464.755,Z 279.421,A 0.000,B 0.000,C 90.000,E1 111.791} C_DIS
LIN {X 0.077,Y -460.875,Z 279.409,A 0.000,B 0.000,C 90.000,E1 109.577} C_DIS
LIN {X 0.125,Y -459.351,Z 279.404,A 0.000,B 0.000,C 90.000,E1 108.671} C_DIS
LIN {X 0.086,Y -459.346,Z 279.404,A 0.000,B 0.000,C 90.000,E1 108.671} C_DIS
LIN {X -0.056,Y -467.911,Z 279.382,A 0.000,B 0.000,C 90.000,E1 104.828} C_DIS
LIN {X -0.029,Y -475.482,Z 279.358,A 0.000,B 0.000,C 90.000,E1 100.433} C_DIS
LIN {X -0.190,Y -476.125,Z 279.356,A 0.000,B 0.000,C 90.000,E1 100.141} C_DIS
LIN {X 0.093,Y -482.042,Z 279.330,A 0.000,B 0.000,C 90.000,E1 95.454} C_DIS
LIN {X -0.116,Y -485.475,Z 279.305,A 0.000,B 0.000,C 90.000,E1 90.859} C_DIS
LIN {X 0.103,Y -485.873,Z 279.288,A 0.000,B 0.000,C 90.000,E1 87.764} C_DIS
LIN {X -0.084,Y -486.386,Z 279.281,A 0.000,B 0.000,C 90.000,E1 86.560} C_DIS
LIN {X 0.226,Y -486.363,Z 279.279,A 0.000,B 0.000,C 90.000,E1 86.216} C_DIS
LIN {X -0.171,Y -484.690,Z 279.254,A 0.000,B 0.000,C 90.000,E1 81.659} C_DIS
LIN {X -0.156,Y -483.695,Z 279.248,A 0.000,B 0.000,C 90.000,E1 80.735} C_DIS
LIN {X 0.208,Y -480.626,Z 279.228,A 0.000,B 0.000,C 90.000,E1 76.992} C_DIS
LIN {X 0.066,Y -480.303,Z 279.226,A 0.000,B 0.000,C 90.000,E1 76.700} C_DIS
LIN {X -0.030,Y -474.123,Z 279.200,A 0.000,B 0.000,C 90.000,E1 72.054} C_DIS
LIN {X 0.178,Y -471.469,Z 279.193,A 0.000,B 0.000,C 90.000,E1 70.678} C_DIS
LIN {X 0.138,Y -471.473,Z 279.193,A 0.000,B 0.000,C 90.000,E1 70.678} C_DIS
LIN {X 0.180,Y -476.699,Z 279.181,A 0.000,B 0.000,C 90.000,E1 68.592} C_DIS
LIN {X 0.089,Y -481.568,Z 279.171,A 0.000,B 0.000,C 90.000,E1 66.741} C_DIS
LIN {X -0.150,Y -486.580,Z 279.161,A 0.000,B 0.000,C 90.000,E1 64.921} C_DIS
LIN {X 0.173,Y -492.493,Z 279.149,A 0.000,B 0.000,C 90.000,E1 62.743} C_DIS
LIN {X -0.223,Y -498.540,Z 279.137,A 0.000,B 0.000,C 90.000,E1 60.667} C_DIS
LIN {X -0.277,Y -503.802,Z 279.127,A 0.000,B 0.000,C 90.000,E1 58.869} C_DIS
LIN {X -0.160,Y -507.348,Z 279.120,A 0.000,B 0.000,C 90.000,E1 57.661} C_DIS
LIN {X 0.287,Y -510.754,Z 279.114,A 0.000,B 0.000,C 90.000,E1 56.421} C_DIS
LIN {X 0.076,Y -514.169,Z 279.107,A 0.000,B 0.000,C 90.000,E1 55.261} C_DIS
LIN {X 0.136,Y -518.045,Z 279.099,A 0.000,B 0.000,C 90.000,E1 53.783} C_DIS
LIN {X -0.100,Y -520.971,Z 279.092,A 0.000,B 0.000,C 90.000,E1 52.637} C_DIS
LIN {X 0.072,Y -523.045,Z 279.088,A 0.000,B 0.000,C 90.000,E1 51.743} C_DIS
LIN {X 0.199,Y -526.168,Z 279.079,A 0.000,B 0.000,C 90.000,E1 50.275} C_DIS
LIN {X 0.004,Y -528.402,Z 279.073,A 0.000,B 0.000,C 90.000,E1 49.138} C_DIS
LIN {X -0.160,Y -530.334,Z 279.067,A 0.000,B 0.000,C 90.000,E1 48.000} C_DIS
LIN {X 0.059,Y -531.927,Z 279.060,A 0.000,B 0.000,C 90.000,E1 46.824} C_DIS
LIN {X -0.043,Y -532.921,Z 279.055,A 0.000,B 0.000,C 90.000,E1 45.972} C_DIS
LIN {X 0.236,Y -533.736,Z 279.051,A 0.000,B 0.000,C 90.000,E1 45.081} C_DIS
LIN {X -0.289,Y -534.669,Z 279.043,A 0.000,B 0.000,C 90.000,E1 43.704} C_DIS
LIN {X -0.022,Y -535.202,Z 279.035,A 0.000,B 0.000,C 90.000,E1 42.243} C_DIS
LIN {X -0.085,Y -535.385,Z 279.030,A 0.000,B 0.000,C 90.000,E1 41.391} C_DIS
LIN {X -0.152,Y -535.334,Z 279.024,A 0.000,B 0.000,C 90.000,E1 40.253} C_DIS
LIN {X -0.224,Y -535.071,Z 279.017,A 0.000,B 0.000,C 90.000,E1 39.116} C_DIS
LIN {X 0.107,Y -534.472,Z 279.011,A 0.000,B 0.000,C 90.000,E1 37.935} C_DIS
LIN {X 0.097,Y -533.548,Z 279.003,A 0.000,B 0.000,C 90.000,E1 36.503} C_DIS
LIN {X -0.241,Y -532.318,Z 278.995,A 0.000,B 0.000,C 90.000,E1 35.105} C_DIS
LIN {X -0.173,Y -530.565,Z 278.985,A 0.000,B 0.000,C 90.000,E1 33.372} C_DIS
LIN {X -0.129,Y -528.957,Z 278.977,A 0.000,B 0.000,C 90.000,E1 31.926} C_DIS
LIN {X 0.052,Y -527.342,Z 278.969,A 0.000,B 0.000,C 90.000,E1 30.463} C_DIS
LIN {X -0.109,Y -525.328,Z 278.960,A 0.000,B 0.000,C 90.000,E1 28.743} C_DIS
LIN {X 0.209,Y -523.697,Z 278.952,A 0.000,B 0.000,C 90.000,E1 27.257} C_DIS
LIN {X -0.053,Y -521.711,Z 278.942,A 0.000,B 0.000,C 90.000,E1 25.540} C_DIS
LIN {X -0.213,Y -519.654,Z 278.931,A 0.000,B 0.000,C 90.000,E1 23.515} C_DIS
LIN {X 0.174,Y -517.937,Z 278.921,A 0.000,B 0.000,C 90.000,E1 21.716} C_DIS
LIN {X -0.022,Y -516.124,Z 278.909,A 0.000,B 0.000,C 90.000,E1 19.685} C_DIS
LIN {X -0.005,Y -514.338,Z 278.896,A 0.000,B 0.000,C 90.000,E1 17.330} C_DIS
LIN {X 0.190,Y -512.922,Z 278.885,A 0.000,B 0.000,C 90.000,E1 15.245} C_DIS
LIN {X 0.130,Y -511.959,Z 278.875,A 0.000,B 0.000,C 90.000,E1 13.480} C_DIS
LIN {X 0.024,Y -511.073,Z 278.864,A 0.000,B 0.000,C 90.000,E1 11.422} C_DIS
LIN {X -0.219,Y -510.448,Z 278.852,A 0.000,B 0.000,C 90.000,E1 9.378} C_DIS
LIN {X 0.211,Y -510.080,Z 278.837,A 0.000,B 0.000,C 90.000,E1 6.663} C_DIS
LIN {X 0.066,Y -510.283,Z 278.822,A 0.000,B 0.000,C 90.000,E1 4.012} C_DIS
LIN {X 0.240,Y -511.132,Z 278.806,A 0.000,B 0.000,C 90.000,E1 1.031} C_DIS
LIN {X -0.135,Y -512.441,Z 278.792,A 0.000,B 0.000,C 90.000,E1 358.625} C_DIS
LIN {X -0.221,Y -514.302,Z 278.779,A 0.000,B 0.000,C 90.000,E1 356.274} C_DIS
LIN {X -0.139,Y -516.348,Z 278.768,A 0.000,B 0.000,C 90.000,E1 354.204} C_DIS
LIN {X -0.069,Y -520.486,Z 278.750,A 0.000,B 0.000,C 90.000,E1 350.971} C_DIS
LIN {X -0.014,Y -525.442,Z 278.735,A 0.000,B 0.000,C 90.000,E1 348.342} C_DIS
LIN {X -0.173,Y -531.798,Z 278.721,A 0.000,B 0.000,C 90.000,E1 345.755} C_DIS
LIN {X -0.116,Y -536.900,Z 278.710,A 0.000,B 0.000,C 90.000,E1 343.740} C_DIS
LIN {X -0.302,Y -542.354,Z 278.699,A 0.000,B 0.000,C 90.000,E1 341.764} C_DIS
LIN {X -0.191,Y -550.161,Z 278.684,A 0.000,B 0.000,C 90.000,E1 339.209} C_DIS
LIN {X 0.291,Y -557.652,Z 278.672,A 0.000,B 0.000,C 90.000,E1 336.922} C_DIS
LIN {X -0.127,Y -564.390,Z 278.661,A 0.000,B 0.000,C 90.000,E1 335.025} C_DIS
LIN {X -0.044,Y -572.355,Z 278.649,A 0.000,B 0.000,C 90.000,E1 332.820} C_DIS
LIN {X 0.078,Y -576.346,Z 278.643,A 0.000,B 0.000,C 90.000,E1 331.719} C_DIS
LIN {X -0.250,Y -580.166,Z 278.637,A 0.000,B 0.000,C 90.000,E1 330.667} C_DIS
LIN {X 0.134,Y -584.793,Z 278.629,A 0.000,B 0.000,C 90.000,E1 329.282} C_DIS
LIN {X 0.095,Y -589.307,Z 278.622,A 0.000,B 0.000,C 90.000,E1 327.946} C_DIS
LIN {X 0.054,Y -595.897,Z 278.612,A 0.000,B 0.000,C 90.000,E1 326.087} C_DIS
LIN {X 0.032,Y -600.800,Z 278.604,A 0.000,B 0.000,C 90.000,E1 324.769} C_DIS
LIN {X 0.187,Y -604.770,Z 278.599,A 0.000,B 0.000,C 90.000,E1 323.703} C_DIS
LIN {X -0.086,Y -608.549,Z 278.593,A 0.000,B 0.000,C 90.000,E1 322.683} C_DIS
LIN {X -0.016,Y -613.001,Z 278.585,A 0.000,B 0.000,C 90.000,E1 321.376} C_DIS
LIN {X -0.049,Y -618.093,Z 278.577,A 0.000,B 0.000,C 90.000,E1 319.828} C_DIS
LIN {X 0.270,Y -623.651,Z 278.567,A 0.000,B 0.000,C 90.000,E1 318.000} C_DIS
LIN {X 0.052,Y -627.401,Z 278.560,A 0.000,B 0.000,C 90.000,E1 316.743} C_DIS
LIN {X -0.107,Y -631.066,Z 278.553,A 0.000,B 0.000,C 90.000,E1 315.486} C_DIS
LIN {X 0.234,Y -634.660,Z 278.546,A 0.000,B 0.000,C 90.000,E1 314.190} C_DIS
LIN {X 0.196,Y -638.073,Z 278.539,A 0.000,B 0.000,C 90.000,E1 312.933} C_DIS
LIN {X 0.299,Y -640.685,Z 278.533,A 0.000,B 0.000,C 90.000,E1 311.919} C_DIS
LIN {X 0.011,Y -643.011,Z 278.528,A 0.000,B 0.000,C 90.000,E1 310.943} C_DIS
LIN {X 0.171,Y -645.061,Z 278.522,A 0.000,B 0.000,C 90.000,E1 309.930} C_DIS
LIN {X -0.068,Y -646.893,Z 278.516,A 0.000,B 0.000,C 90.000,E1 308.955} C_DIS
LIN {X -0.260,Y -648.912,Z 278.510,A 0.000,B 0.000,C 90.000,E1 307.729} C_DIS
LIN {X 0.054,Y -650.290,Z 278.504,A 0.000,B 0.000,C 90.000,E1 306.710} C_DIS
LIN {X 0.081,Y -651.109,Z 278.500,A 0.000,B 0.000,C 90.000,E1 305.964} C_DIS
LIN {X -0.027,Y -651.593,Z 278.496,A 0.000,B 0.000,C 90.000,E1 305.231} C_DIS
LIN {X 0.026,Y -651.844,Z 278.492,A 0.000,B 0.000,C 90.000,E1 304.485} C_DIS
LIN {X 0.072,Y -651.997,Z 278.485,A 0.000,B 0.000,C 90.000,E1 303.245} C_DIS
LIN {X 0.138,Y -651.752,Z 278.481,A 0.000,B 0.000,C 90.000,E1 302.498} C_DIS
LIN {X 0.201,Y -651.204,Z 278.477,A 0.000,B 0.000,C 90.000,E1 301.750} C_DIS
LIN {X -0.210,Y -650.009,Z 278.471,A 0.000,B 0.000,C 90.000,E1 300.797} C_DIS
LIN {X -0.174,Y -648.726,Z 278.467,A 0.000,B 0.000,C 90.000,E1 300.050} C_DIS
LIN {X 0.174,Y -646.626,Z 278.461,A 0.000,B 0.000,C 90.000,E1 299.027} C_DIS
LIN {X 0.320,Y -643.671,Z 278.454,A 0.000,B 0.000,C 90.000,E1 297.769} C_DIS
LIN {X -0.114,Y -639.874,Z 278.446,A 0.000,B 0.000,C 90.000,E1 296.309} C_DIS
LIN {X 0.074,Y -637.859,Z 278.442,A 0.000,B 0.000,C 90.000,E1 295.540} C_DIS
LIN {X 0.153,Y -633.168,Z 278.432,A 0.000,B 0.000,C 90.000,E1 293.770} C_DIS
LIN {X -0.157,Y -629.140,Z 278.424,A 0.000,B 0.000,C 90.000,E1 292.280} C_DIS
LIN {X 0.037,Y -624.614,Z 278.414,A 0.000,B 0.000,C 90.000,E1 290.482} C_DIS
LIN {X 0.239,Y -619.588,Z 278.402,A 0.000,B 0.000,C 90.000,E1 288.417} C_DIS
LIN {X -0.067,Y -614.955,Z 278.391,A 0.000,B 0.000,C 90.000,E1 286.386} C_DIS
LIN {X 0.199,Y -609.948,Z 278.377,A 0.000,B 0.000,C 90.000,E1 283.772} C_DIS
LIN {X 0.004,Y -604.447,Z 278.356,A 0.000,B 0.000,C 90.000,E1 280.141} C_DIS
LIN {X 0.134,Y -600.924,Z 278.337,A 0.000,B 0.000,C 90.000,E1 276.720} C_DIS
LIN {X 0.210,Y -598.989,Z 278.320,A 0.000,B 0.000,C 90.000,E1 273.555} C_DIS
LIN {X -0.125,Y -598.412,Z 278.304,A 0.000,B 0.000,C 90.000,E1 270.688} C_DIS
LIN {X -0.124,Y -598.782,Z 278.289,A 0.000,B 0.000,C 90.000,E1 268.051} C_DIS
LIN {X 0.047,Y -599.858,Z 278.277,A 0.000,B 0.000,C 90.000,E1 265.927} C_DIS
LIN {X 0.291,Y -601.551,Z 278.266,A 0.000,B 0.000,C 90.000,E1 263.799} C_DIS
LIN {X 0.064,Y -604.431,Z 278.251,A 0.000,B 0.000,C 90.000,E1 261.197} C_DIS
LIN {X -0.202,Y -607.665,Z 278.238,A 0.000,B 0.000,C 90.000,E1 258.870} C_DIS
LIN {X -0.218,Y -610.562,Z 278.228,A 0.000,B 0.000,C 90.000,E1 257.048} C_DIS
LIN {X -0.272,Y -612.574,Z 278.221,A 0.000,B 0.000,C 90.000,E1 255.755} C_DIS
LIN {X -0.064,Y -614.191,Z 278.215,A 0.000,B 0.000,C 90.000,E1 254.700} C_DIS
LIN {X -0.032,Y -615.277,Z 278.211,A 0.000,B 0.000,C 90.000,E1 253.921} C_DIS
LIN {X 0.016,Y -616.092,Z 278.206,A 0.000,B 0.000,C 90.000,E1 253.142} C_DIS
LIN {X -0.165,Y -616.882,Z 278.201,A 0.000,B 0.000,C 90.000,E1 252.127} C_DIS
LIN {X -0.387,Y -617.585,Z 278.194,A 0.000,B 0.000,C 90.000,E1 250.859} C_DIS
LIN {X -0.147,Y -617.800,Z 278.188,A 0.000,B 0.000,C 90.000,E1 249.806} C_DIS
LIN {X -0.112,Y -617.603,Z 278.182,A 0.000,B 0.000,C 90.000,E1 248.773} C_DIS
LIN {X 0.162,Y -617.158,Z 278.178,A 0.000,B 0.000,C 90.000,E1 247.975} C_DIS
LIN {X -0.140,Y -616.529,Z 278.173,A 0.000,B 0.000,C 90.000,E1 247.230} C_DIS
LIN {X 0.116,Y -615.616,Z 278.169,A 0.000,B 0.000,C 90.000,E1 246.433} C_DIS
LIN {X 0.044,Y -614.457,Z 278.165,A 0.000,B 0.000,C 90.000,E1 245.665} C_DIS
LIN {X -0.290,Y -613.048,Z 278.161,A 0.000,B 0.000,C 90.000,E1 244.921} C_DIS
LIN {X -0.349,Y -612.035,Z 278.158,A 0.000,B 0.000,C 90.000,E1 244.409} C_DIS
LIN {X 0.063,Y -609.654,Z 278.152,A 0.000,B 0.000,C 90.000,E1 243.332} C_DIS
LIN {X 0.173,Y -607.097,Z 278.146,A 0.000,B 0.000,C 90.000,E1 242.281} C_DIS
LIN {X -0.091,Y -603.683,Z 278.139,A 0.000,B 0.000,C 90.000,E1 241.001} C_DIS
LIN {X 0.170,Y -600.125,Z 278.132,A 0.000,B 0.000,C 90.000,E1 239.665} C_DIS
LIN {X 0.374,Y -596.345,Z 278.124,A 0.000,B 0.000,C 90.000,E1 238.329} C_DIS
LIN {X 0.005,Y -592.382,Z 278.117,A 0.000,B 0.000,C 90.000,E1 237.041} C_DIS
LIN {X -0.103,Y -588.168,Z 278.110,A 0.000,B 0.000,C 90.000,E1 235.722} C_DIS
LIN {X -0.096,Y -582.956,Z 278.101,A 0.000,B 0.000,C 90.000,E1 234.116} C_DIS
LIN {X 0.302,Y -577.092,Z 278.090,A 0.000,B 0.000,C 90.000,E1 232.190} C_DIS
LIN {X -0.195,Y -572.866,Z 278.083,A 0.000,B 0.000,C 90.000,E1 230.884} C_DIS
LIN {X -0.033,Y -568.663,Z 278.075,A 0.000,B 0.000,C 90.000,E1 229.504} C_DIS
LIN {X 0.168,Y -563.558,Z 278.066,A 0.000,B 0.000,C 90.000,E1 227.838} C_DIS
LIN {X -0.166,Y -558.386,Z 278.057,A 0.000,B 0.000,C 90.000,E1 226.215} C_DIS
LIN {X 0.159,Y -553.178,Z 278.047,A 0.000,B 0.000,C 90.000,E1 224.514} C_DIS
LIN {X -0.069,Y -549.693,Z 278.041,A 0.000,B 0.000,C 90.000,E1 223.419} C_DIS
LIN {X -0.312,Y -544.447,Z 278.032,A 0.000,B 0.000,C 90.000,E1 221.757} C_DIS
LIN {X 0.115,Y -540.127,Z 278.024,A 0.000,B 0.000,C 90.000,E1 220.297} C_DIS
LIN {X 0.108,Y -534.861,Z 278.014,A 0.000,B 0.000,C 90.000,E1 218.588} C_DIS
LIN {X 0.079,Y -529.688,Z 278.005,A 0.000,B 0.000,C 90.000,E1 216.870} C_DIS
LIN {X -0.060,Y -524.580,Z 277.995,A 0.000,B 0.000,C 90.000,E1 215.152} C_DIS
LIN {X 0.189,Y -518.812,Z 277.984,A 0.000,B 0.000,C 90.000,E1 213.086} C_DIS
LIN {X 0.011,Y -513.283,Z 277.973,A 0.000,B 0.000,C 90.000,E1 211.052} C_DIS
LIN {X -0.053,Y -507.206,Z 277.959,A 0.000,B 0.000,C 90.000,E1 208.693} C_DIS
LIN {X -0.144,Y -502.226,Z 277.948,A 0.000,B 0.000,C 90.000,E1 206.616} C_DIS
LIN {X -0.085,Y -496.975,Z 277.934,A 0.000,B 0.000,C 90.000,E1 204.207} C_DIS
LIN {X -0.027,Y -493.266,Z 277.924,A 0.000,B 0.000,C 90.000,E1 202.386} C_DIS
LIN {X 0.142,Y -487.524,Z 277.908,A 0.000,B 0.000,C 90.000,E1 199.322} C_DIS
LIN {X 0.094,Y -482.925,Z 277.892,A 0.000,B 0.000,C 90.000,E1 196.567} C_DIS
LIN {X 0.085,Y -478.304,Z 277.875,A 0.000,B 0.000,C 90.000,E1 193.480} C_DIS
LIN {X 0.148,Y -475.505,Z 277.863,A 0.000,B 0.000,C 90.000,E1 191.299} C_DIS
LIN {X -0.191,Y -471.840,Z 277.846,A 0.000,B 0.000,C 90.000,E1 188.219} C_DIS
LIN {X 0.009,Y -469.927,Z 277.835,A 0.000,B 0.000,C 90.000,E1 186.315} C_DIS
LIN {X 0.141,Y -467.585,Z 277.821,A 0.000,B 0.000,C 90.000,E1 183.784} C_DIS
LIN {X 0.141,Y -466.160,Z 277.811,A 0.000,B 0.000,C 90.000,E1 181.892} C_DIS
LIN {X 0.090,Y -464.467,Z 277.797,A 0.000,B 0.000,C 90.000,E1 179.370} C_DIS
LIN {X -0.229,Y -463.411,Z 277.784,A 0.000,B 0.000,C 90.000,E1 177.192} C_DIS
LIN {X -0.078,Y -462.442,Z 277.768,A 0.000,B 0.000,C 90.000,E1 174.318} C_DIS
LIN {X -0.108,Y -462.079,Z 277.754,A 0.000,B 0.000,C 90.000,E1 171.781} C_DIS
LIN {X 0.220,Y -461.989,Z 277.745,A 0.000,B 0.000,C 90.000,E1 170.151} C_DIS
LIN {X 0.175,Y -462.239,Z 277.730,A 0.000,B 0.000,C 90.000,E1 167.297} C_DIS
LIN {X -0.047,Y -462.758,Z 277.717,A 0.000,B 0.000,C 90.000,E1 165.102} C_DIS
LIN {X 0.043,Y -464.046,Z 277.701,A 0.000,B 0.000,C 90.000,E1 162.236} C_DIS
LIN {X -0.228,Y -465.346,Z 277.691,A 0.000,B 0.000,C 90.000,E1 160.369} C_DIS
LIN {X 0.161,Y -467.396,Z 277.677,A 0.000,B 0.000,C 90.000,E1 157.794} C_DIS
LIN {X 0.117,Y -469.885,Z 277.663,A 0.000,B 0.000,C 90.000,E1 155.281} C_DIS
LIN {X -0.110,Y -473.339,Z 277.647,A 0.000,B 0.000,C 90.000,E1 152.487} C_DIS
LIN {X -0.176,Y -476.957,Z 277.633,A 0.000,B 0.000,C 90.000,E1 149.999} C_DIS
LIN {X -0.056,Y -479.903,Z 277.623,A 0.000,B 0.000,C 90.000,E1 148.122} C_DIS
LIN {X -0.088,Y -482.481,Z 277.614,A 0.000,B 0.000,C 90.000,E1 146.580} C_DIS
LIN {X 0.282,Y -485.624,Z 277.604,A 0.000,B 0.000,C 90.000,E1 144.689} C_DIS
LIN {X -0.054,Y -488.819,Z 277.594,A 0.000,B 0.000,C 90.000,E1 142.889} C_DIS
LIN {X -0.007,Y -490.795,Z 277.587,A 0.000,B 0.000,C 90.000,E1 141.662} C_DIS
LIN {X -0.091,Y -493.158,Z 277.579,A 0.000,B 0.000,C 90.000,E1 140.150} C_DIS
LIN {X -0.057,Y -494.826,Z 277.572,A 0.000,B 0.000,C 90.000,E1 138.933} C_DIS
LIN {X 0.004,Y -496.290,Z 277.565,A 0.000,B 0.000,C 90.000,E1 137.715} C_DIS
LIN {X 0.040,Y -496.873,Z 277.562,A 0.000,B 0.000,C 90.000,E1 137.106} C_DIS
LIN {X -0.092,Y -497.521,Z 277.557,A 0.000,B 0.000,C 90.000,E1 136.215} C_DIS
LIN {X -0.212,Y -497.978,Z 277.552,A 0.000,B 0.000,C 90.000,E1 135.324} C_DIS
LIN {X 0.024,Y -498.239,Z 277.547,A 0.000,B 0.000,C 90.000,E1 134.393} C_DIS
LIN {X 0.122,Y -498.089,Z 277.540,A 0.000,B 0.000,C 90.000,E1 133.176} C_DIS
LIN {X 0.005,Y -497.743,Z 277.535,A 0.000,B 0.000,C 90.000,E1 132.285} C_DIS
LIN {X -0.084,Y -497.157,Z 277.530,A 0.000,B 0.000,C 90.000,E1 131.391} C_DIS
LIN {X 0.150,Y -496.321,Z 277.525,A 0.000,B 0.000,C 90.000,E1 130.458} C_DIS
LIN {X -0.091,Y -494.963,Z 277.518,A 0.000,B 0.000,C 90.000,E1 129.277} C_DIS
LIN {X 0.038,Y -493.385,Z 277.511,A 0.000,B 0.000,C 90.000,E1 128.051} C_DIS
LIN {X -0.246,Y -491.632,Z 277.505,A 0.000,B 0.000,C 90.000,E1 126.870} C_DIS
LIN {X 0.226,Y -489.687,Z 277.498,A 0.000,B 0.000,C 90.000,E1 125.598} C_DIS
LIN {X -0.016,Y -487.541,Z 277.491,A 0.000,B 0.000,C 90.000,E1 124.405} C_DIS
LIN {X 0.112,Y -485.293,Z 277.484,A 0.000,B 0.000,C 90.000,E1 123.166} C_DIS
LIN {X -0.023,Y -481.760,Z 277.474,A 0.000,B 0.000,C 90.000,E1 121.337} C_DIS
LIN {X -0.037,Y -478.966,Z 277.466,A 0.000,B 0.000,C 90.000,E1 119.795} C_DIS
LIN {X 0.259,Y -475.440,Z 277.455,A 0.000,B 0.000,C 90.000,E1 117.897} C_DIS
LIN {X 0.041,Y -471.964,Z 277.445,A 0.000,B 0.000,C 90.000,E1 116.052} C_DIS
LIN {X -0.110,Y -467.781,Z 277.433,A 0.000,B 0.000,C 90.000,E1 113.875} C_DIS
LIN {X -0.082,Y -463.764,Z 277.420,A 0.000,B 0.000,C 90.000,E1 111.663} C_DIS
LIN {X -0.152,Y -459.921,Z 277.408,A 0.000,B 0.000,C 90.000,E1 109.450} C_DIS
LIN {X -0.224,Y -458.978,Z 277.405,A 0.000,B 0.000,C 90.000,E1 108.906} C_DIS
LIN {X 0.171,Y -458.979,Z 277.405,A 0.000,B 0.000,C 90.000,E1 108.852} C_DIS
LIN {X -0.226,Y -467.571,Z 277.383,A 0.000,B 0.000,C 90.000,E1 105.009} C_DIS
LIN {X -0.042,Y -468.579,Z 277.380,A 0.000,B 0.000,C 90.000,E1 104.356} C_DIS
LIN {X 0.184,Y -475.804,Z 277.357,A 0.000,B 0.000,C 90.000,E1 100.254} C_DIS
LIN {X 0.023,Y -476.306,Z 277.355,A 0.000,B 0.000,C 90.000,E1 99.962} C_DIS
LIN {X -0.029,Y -481.791,Z 277.331,A 0.000,B 0.000,C 90.000,E1 95.625} C_DIS
LIN {X -0.183,Y -482.171,Z 277.330,A 0.000,B 0.000,C 90.000,E1 95.334} C_DIS
LIN {X 0.232,Y -485.309,Z 277.306,A 0.000,B 0.000,C 90.000,E1 90.974} C_DIS
LIN {X 0.056,Y -485.537,Z 277.304,A 0.000,B 0.000,C 90.000,E1 90.688} C_DIS
LIN {X -0.222,Y -486.320,Z 277.282,A 0.000,B 0.000,C 90.000,E1 86.731} C_DIS
LIN {X -0.087,Y -486.304,Z 277.278,A 0.000,B 0.000,C 90.000,E1 86.102} C_DIS
LIN {X 0.118,Y -484.696,Z 277.254,A 0.000,B 0.000,C 90.000,E1 81.781} C_DIS
LIN {X -0.014,Y -484.599,Z 277.253,A 0.000,B 0.000,C 90.000,E1 81.489} C_DIS
LIN {X -0.134,Y -480.533,Z 277.227,A 0.000,B 0.000,C 90.000,E1 76.881} C_DIS
LIN {X 0.229,Y -474.284,Z 277.201,A 0.000,B 0.000,C 90.000,E1 72.181} C_DIS
LIN {X 0.197,Y -473.845,Z 277.199,A 0.000,B 0.000,C 90.000,E1 71.873} C_DIS
LIN {X 0.156,Y -471.126,Z 277.192,A 0.000,B 0.000,C 90.000,E1 70.496} C_DIS
LIN {X 0.116,Y -471.131,Z 277.192,A 0.000,B 0.000,C 90.000,E1 70.496} C_DIS
LIN {X -0.026,Y -475.476,Z 277.182,A 0.000,B 0.000,C 90.000,E1 68.773} C_DIS
LIN {X -0.143,Y -480.359,Z 277.172,A 0.000,B 0.000,C 90.000,E1 66.922} C_DIS
LIN {X 0.033,Y -485.348,Z 277.161,A 0.000,B 0.000,C 90.000,E1 65.049} C_DIS
LIN {X 0.157,Y -492.956,Z 277.146,A 0.000,B 0.000,C 90.000,E1 62.281} C_DIS
LIN {X -0.225,Y -498.976,Z 277.134,A 0.000,B 0.000,C 90.000,E1 60.205} C_DIS
LIN {X 0.118,Y -503.409,Z 277.126,A 0.000,B 0.000,C 90.000,E1 58.663} C_DIS
LIN {X 0.125,Y -507.786,Z 277.118,A 0.000,B 0.000,C 90.000,E1 57.168} C_DIS
LIN {X 0.123,Y -512.914,Z 277.108,A 0.000,B 0.000,C 90.000,E1 55.388} C_DIS
LIN {X 0.234,Y -516.045,Z 277.101,A 0.000,B 0.000,C 90.000,E1 54.196} C_DIS
LIN {X -0.027,Y -519.022,Z 277.095,A 0.000,B 0.000,C 90.000,E1 53.050} C_DIS
LIN {X -0.247,Y -521.846,Z 277.088,A 0.000,B 0.000,C 90.000,E1 51.904} C_DIS
LIN {X -0.148,Y -525.003,Z 277.080,A 0.000,B 0.000,C 90.000,E1 50.436} C_DIS
LIN {X 0.036,Y -527.226,Z 277.074,A 0.000,B 0.000,C 90.000,E1 49.256} C_DIS
LIN {X 0.200,Y -529.188,Z 277.067,A 0.000,B 0.000,C 90.000,E1 48.081} C_DIS
LIN {X 0.072,Y -530.408,Z 277.062,A 0.000,B 0.000,C 90.000,E1 47.229} C_DIS
LIN {X -0.046,Y -531.494,Z 277.058,A 0.000,B 0.000,C 90.000,E1 46.377} C_DIS
LIN {X -0.198,Y -532.625,Z 277.051,A 0.000,B 0.000,C 90.000,E1 45.243} C_DIS
LIN {X -0.266,Y -533.070,Z 277.048,A 0.000,B 0.000,C 90.000,E1 44.676} C_DIS
LIN {X 0.013,Y -533.596,Z 277.043,A 0.000,B 0.000,C 90.000,E1 43.785} C_DIS
LIN {X -0.134,Y -534.114,Z 277.035,A 0.000,B 0.000,C 90.000,E1 42.366} C_DIS
LIN {X -0.213,Y -534.307,Z 277.031,A 0.000,B 0.000,C 90.000,E1 41.515} C_DIS
LIN {X 0.112,Y -534.305,Z 277.026,A 0.000,B 0.000,C 90.000,E1 40.620} C_DIS
LIN {X 0.024,Y -534.088,Z 277.019,A 0.000,B 0.000,C 90.000,E1 39.483} C_DIS
LIN {X 0.010,Y -533.593,Z 277.013,A 0.000,B 0.000,C 90.000,E1 38.338} C_DIS
LIN {X 0.309,Y -532.458,Z 277.003,A 0.000,B 0.000,C 90.000,E1 36.583} C_DIS
LIN {X -0.046,Y -531.209,Z 276.995,A 0.000,B 0.000,C 90.000,E1 35.185} C_DIS
LIN {X 0.000,Y -529.437,Z 276.986,A 0.000,B 0.000,C 90.000,E1 33.452} C_DIS
LIN {X 0.028,Y -527.815,Z 276.978,A 0.000,B 0.000,C 90.000,E1 32.005} C_DIS
LIN {X 0.192,Y -526.152,Z 276.970,A 0.000,B 0.000,C 90.000,E1 30.541} C_DIS
LIN {X -0.134,Y -524.445,Z 276.962,A 0.000,B 0.000,C 90.000,E1 29.127} C_DIS
LIN {X -0.153,Y -522.440,Z 276.952,A 0.000,B 0.000,C 90.000,E1 27.385} C_DIS
LIN {X 0.252,Y -520.434,Z 276.942,A 0.000,B 0.000,C 90.000,E1 25.591} C_DIS
LIN {X 0.192,Y -518.068,Z 276.929,A 0.000,B 0.000,C 90.000,E1 23.259} C_DIS
LIN {X -0.134,Y -516.340,Z 276.920,A 0.000,B 0.000,C 90.000,E1 21.535} C_DIS
LIN {X 0.242,Y -514.310,Z 276.907,A 0.000,B 0.000,C 90.000,E1 19.141} C_DIS
LIN {X 0.055,Y -512.556,Z 276.893,A 0.000,B 0.000,C 90.000,E1 16.804} C_DIS
LIN {X 0.229,Y -510.703,Z 276.877,A 0.000,B 0.000,C 90.000,E1 13.828} C_DIS
LIN {X 0.045,Y -509.583,Z 276.864,A 0.000,B 0.000,C 90.000,E1 11.478} C_DIS
LIN {X 0.263,Y -508.946,Z 276.852,A 0.000,B 0.000,C 90.000,E1 9.378} C_DIS
LIN {X 0.135,Y -508.530,Z 276.837,A 0.000,B 0.000,C 90.000,E1 6.720} C_DIS
LIN {X -0.098,Y -508.687,Z 276.823,A 0.000,B 0.000,C 90.000,E1 4.073} C_DIS
LIN {X 0.141,Y -509.386,Z 276.808,A 0.000,B 0.000,C 90.000,E1 1.375} C_DIS
LIN {X -0.247,Y -511.013,Z 276.791,A 0.000,B 0.000,C 90.000,E1 358.339} C_DIS
LIN {X 0.084,Y -513.194,Z 276.776,A 0.000,B 0.000,C 90.000,E1 355.641} C_DIS
LIN {X -0.254,Y -514.663,Z 276.768,A 0.000,B 0.000,C 90.000,E1 354.204} C_DIS
LIN {X -0.263,Y -519.320,Z 276.748,A 0.000,B 0.000,C 90.000,E1 350.679} C_DIS
LIN {X 0.259,Y -523.797,Z 276.735,A 0.000,B 0.000,C 90.000,E1 348.285} C_DIS
LIN {X 0.045,Y -530.229,Z 276.721,A 0.000,B 0.000,C 90.000,E1 345.700} C_DIS
LIN {X 0.019,Y -534.606,Z 276.711,A 0.000,B 0.000,C 90.000,E1 343.976} C_DIS
LIN {X -0.219,Y -540.071,Z 276.700,A 0.000,B 0.000,C 90.000,E1 342.000} C_DIS
LIN {X 0.084,Y -548.697,Z 276.684,A 0.000,B 0.000,C 90.000,E1 339.135} C_DIS
LIN {X -0.192,Y -556.209,Z 276.672,A 0.000,B 0.000,C 90.000,E1 336.922} C_DIS
LIN {X 0.061,Y -561.982,Z 276.662,A 0.000,B 0.000,C 90.000,E1 335.229} C_DIS
LIN {X -0.180,Y -569.976,Z 276.650,A 0.000,B 0.000,C 90.000,E1 333.050} C_DIS
LIN {X 0.263,Y -575.020,Z 276.643,A 0.000,B 0.000,C 90.000,E1 331.641} C_DIS
LIN {X -0.078,Y -578.856,Z 276.637,A 0.000,B 0.000,C 90.000,E1 330.589} C_DIS
LIN {X 0.289,Y -583.531,Z 276.629,A 0.000,B 0.000,C 90.000,E1 329.203} C_DIS
LIN {X 0.233,Y -588.062,Z 276.622,A 0.000,B 0.000,C 90.000,E1 327.867} C_DIS
LIN {X 0.170,Y -594.675,Z 276.611,A 0.000,B 0.000,C 90.000,E1 326.008} C_DIS
LIN {X 0.371,Y -600.621,Z 276.602,A 0.000,B 0.000,C 90.000,E1 324.402} C_DIS
LIN {X -0.316,Y -604.556,Z 276.597,A 0.000,B 0.000,C 90.000,E1 323.417} C_DIS
LIN {X -0.113,Y -608.250,Z 276.591,A 0.000,B 0.000,C 90.000,E1 322.351} C_DIS
LIN {X 0.039,Y -611.818,Z 276.585,A 0.000,B 0.000,C 90.000,E1 321.295} C_DIS
LIN {X -0.015,Y -616.913,Z 276.576,A 0.000,B 0.000,C 90.000,E1 319.747} C_DIS
LIN {X 0.279,Y -622.503,Z 276.566,A 0.000,B 0.000,C 90.000,E1 317.919} C_DIS
LIN {X 0.042,Y -626.336,Z 276.559,A 0.000,B 0.000,C 90.000,E1 316.662} C_DIS
LIN {X -0.135,Y -629.968,Z 276.552,A 0.000,B 0.000,C 90.000,E1 315.405} C_DIS
LIN {X 0.187,Y -633.558,Z 276.545,A 0.000,B 0.000,C 90.000,E1 314.109} C_DIS
LIN {X 0.030,Y -637.629,Z 276.537,A 0.000,B 0.000,C 90.000,E1 312.609} C_DIS
LIN {X 0.217,Y -639.531,Z 276.533,A 0.000,B 0.000,C 90.000,E1 311.838} C_DIS
LIN {X -0.087,Y -641.837,Z 276.527,A 0.000,B 0.000,C 90.000,E1 310.862} C_DIS
LIN {X 0.054,Y -643.824,Z 276.521,A 0.000,B 0.000,C 90.000,E1 309.850} C_DIS
LIN {X -0.116,Y -645.192,Z 276.517,A 0.000,B 0.000,C 90.000,E1 309.116} C_DIS
LIN {X 0.065,Y -647.232,Z 276.510,A 0.000,B 0.000,C 90.000,E1 307.855} C_DIS
LIN {X -0.036,Y -648.633,Z 276.505,A 0.000,B 0.000,C 90.000,E1 306.870} C_DIS
LIN {X -0.165,Y -649.476,Z 276.501,A 0.000,B 0.000,C 90.000,E1 306.137} C_DIS
LIN {X -0.142,Y -650.016,Z 276.497,A 0.000,B 0.000,C 90.000,E1 305.391} C_DIS
LIN {X -0.200,Y -650.348,Z 276.491,A 0.000,B 0.000,C 90.000,E1 304.405} C_DIS
LIN {X 0.283,Y -650.467,Z 276.486,A 0.000,B 0.000,C 90.000,E1 303.372} C_DIS
LIN {X -0.216,Y -650.283,Z 276.481,A 0.000,B 0.000,C 90.000,E1 302.673} C_DIS
LIN {X 0.296,Y -650.035,Z 276.479,A 0.000,B 0.000,C 90.000,E1 302.133} C_DIS
LIN {X -0.003,Y -649.319,Z 276.475,A 0.000,B 0.000,C 90.000,E1 301.416} C_DIS
LIN {X -0.051,Y -648.702,Z 276.472,A 0.000,B 0.000,C 90.000,E1 300.924} C_DIS
LIN {X 0.054,Y -647.009,Z 276.466,A 0.000,B 0.000,C 90.000,E1 299.922} C_DIS
LIN {X -0.184,Y -644.845,Z 276.461,A 0.000,B 0.000,C 90.000,E1 298.949} C_DIS
LIN {X -0.072,Y -641.860,Z 276.454,A 0.000,B 0.000,C 90.000,E1 297.692} C_DIS
LIN {X -0.034,Y -638.698,Z 276.447,A 0.000,B 0.000,C 90.000,E1 296.437} C_DIS
LIN {X 0.195,Y -636.024,Z 276.441,A 0.000,B 0.000,C 90.000,E1 295.412} C_DIS
LIN {X 0.228,Y -631.336,Z 276.432,A 0.000,B 0.000,C 90.000,E1 293.643} C_DIS
LIN {X -0.107,Y -626.629,Z 276.422,A 0.000,B 0.000,C 90.000,E1 291.897} C_DIS
LIN {X 0.026,Y -622.807,Z 276.413,A 0.000,B 0.000,C 90.000,E1 290.355} C_DIS
LIN {X -0.061,Y -617.217,Z 276.400,A 0.000,B 0.000,C 90.000,E1 288.055} C_DIS
LIN {X -0.161,Y -611.674,Z 276.386,A 0.000,B 0.000,C 90.000,E1 285.481} C_DIS
LIN {X -0.247,Y -607.803,Z 276.374,A 0.000,B 0.000,C 90.000,E1 283.411} C_DIS
LIN {X 0.310,Y -602.851,Z 276.356,A 0.000,B 0.000,C 90.000,E1 279.962} C_DIS
LIN {X -0.317,Y -599.391,Z 276.337,A 0.000,B 0.000,C 90.000,E1 276.606} C_DIS
LIN {X -0.168,Y -597.315,Z 276.315,A 0.000,B 0.000,C 90.000,E1 272.636} C_DIS
LIN {X -0.216,Y -597.020,Z 276.300,A 0.000,B 0.000,C 90.000,E1 270.000} C_DIS
LIN {X -0.134,Y -598.124,Z 276.281,A 0.000,B 0.000,C 90.000,E1 266.560} C_DIS
LIN {X 0.287,Y -599.905,Z 276.268,A 0.000,B 0.000,C 90.000,E1 264.147} C_DIS
LIN {X -0.004,Y -602.673,Z 276.253,A 0.000,B 0.000,C 90.000,E1 261.546} C_DIS
LIN {X 0.270,Y -605.860,Z 276.240,A 0.000,B 0.000,C 90.000,E1 259.162} C_DIS
LIN {X -0.179,Y -609.150,Z 276.228,A 0.000,B 0.000,C 90.000,E1 257.117} C_DIS
LIN {X -0.117,Y -611.182,Z 276.221,A 0.000,B 0.000,C 90.000,E1 255.811} C_DIS
LIN {X 0.074,Y -612.788,Z 276.215,A 0.000,B 0.000,C 90.000,E1 254.755} C_DIS
LIN {X -0.148,Y -614.221,Z 276.210,A 0.000,B 0.000,C 90.000,E1 253.740} C_DIS
LIN {X -0.111,Y -615.006,Z 276.205,A 0.000,B 0.000,C 90.000,E1 252.960} C_DIS
LIN {X -0.064,Y -615.592,Z 276.201,A 0.000,B 0.000,C 90.000,E1 252.181} C_DIS
LIN {X -0.302,Y -616.311,Z 276.194,A 0.000,B 0.000,C 90.000,E1 250.913} C_DIS
LIN {X -0.289,Y -616.502,Z 276.188,A 0.000,B 0.000,C 90.000,E1 249.880} C_DIS
LIN {X -0.027,Y -616.436,Z 276.184,A 0.000,B 0.000,C 90.000,E1 249.082} C_DIS
LIN {X 0.236,Y -616.096,Z 276.180,A 0.000,B 0.000,C 90.000,E1 248.284} C_DIS
LIN {X -0.103,Y -615.269,Z 276.174,A 0.000,B 0.000,C 90.000,E1 247.283} C_DIS
LIN {X 0.143,Y -614.406,Z 276.169,A 0.000,B 0.000,C 90.000,E1 246.485} C_DIS
LIN {X -0.190,Y -613.254,Z 276.165,A 0.000,B 0.000,C 90.000,E1 245.741} C_DIS
LIN {X 0.242,Y -611.347,Z 276.159,A 0.000,B 0.000,C 90.000,E1 244.665} C_DIS
LIN {X 0.135,Y -609.665,Z 276.155,A 0.000,B 0.000,C 90.000,E1 243.896} C_DIS
LIN {X -0.030,Y -607.193,Z 276.149,A 0.000,B 0.000,C 90.000,E1 242.871} C_DIS
LIN {X -0.003,Y -603.875,Z 276.142,A 0.000,B 0.000,C 90.000,E1 241.563} C_DIS
LIN {X -0.028,Y -600.375,Z 276.135,A 0.000,B 0.000,C 90.000,E1 240.255} C_DIS
LIN {X -0.036,Y -597.449,Z 276.129,A 0.000,B 0.000,C 90.000,E1 239.203} C_DIS
LIN {X 0.220,Y -594.380,Z 276.123,A 0.000,B 0.000,C 90.000,E1 238.122} C_DIS
LIN {X -0.065,Y -591.198,Z 276.117,A 0.000,B 0.000,C 90.000,E1 237.089} C_DIS
LIN {X 0.162,Y -586.066,Z 276.108,A 0.000,B 0.000,C 90.000,E1 235.468} C_DIS
LIN {X -0.183,Y -580.036,Z 276.098,A 0.000,B 0.000,C 90.000,E1 233.623} C_DIS
LIN {X -0.167,Y -575.898,Z 276.090,A 0.000,B 0.000,C 90.000,E1 232.271} C_DIS
LIN {X -0.184,Y -570.785,Z 276.081,A 0.000,B 0.000,C 90.000,E1 230.642} C_DIS
LIN {X -0.109,Y -567.461,Z 276.075,A 0.000,B 0.000,C 90.000,E1 229.542} C_DIS
LIN {X 0.056,Y -562.347,Z 276.066,A 0.000,B 0.000,C 90.000,E1 227.877} C_DIS
LIN {X 0.071,Y -557.139,Z 276.057,A 0.000,B 0.000,C 90.000,E1 226.215} C_DIS
LIN {X -0.026,Y -551.936,Z 276.048,A 0.000,B 0.000,C 90.000,E1 224.555} C_DIS
LIN {X 0.121,Y -548.415,Z 276.041,A 0.000,B 0.000,C 90.000,E1 223.419} C_DIS
LIN {X -0.152,Y -543.154,Z 276.032,A 0.000,B 0.000,C 90.000,E1 221.757} C_DIS
LIN {X 0.263,Y -537.942,Z 276.022,A 0.000,B 0.000,C 90.000,E1 220.011} C_DIS
LIN {X 0.211,Y -532.681,Z 276.013,A 0.000,B 0.000,C 90.000,E1 218.302} C_DIS
LIN {X 0.137,Y -527.510,Z 276.003,A 0.000,B 0.000,C 90.000,E1 216.583} C_DIS
LIN {X -0.052,Y -522.438,Z 275.994,A 0.000,B 0.000,C 90.000,E1 214.865} C_DIS
LIN {X 0.204,Y -517.504,Z 275.984,A 0.000,B 0.000,C 90.000,E1 213.086} C_DIS
LIN {X -0.008,Y -511.963,Z 275.973,A 0.000,B 0.000,C 90.000,E1 211.052} C_DIS
LIN {X -0.110,Y -505.896,Z 275.959,A 0.000,B 0.000,C 90.000,E1 208.693} C_DIS
LIN {X -0.234,Y -500.911,Z 275.948,A 0.000,B 0.000,C 90.000,E1 206.616} C_DIS
LIN {X 0.184,Y -496.299,Z 275.936,A 0.000,B 0.000,C 90.000,E1 204.463} C_DIS
LIN {X -0.183,Y -491.974,Z 275.924,A 0.000,B 0.000,C 90.000,E1 202.386} C_DIS
LIN {X -0.079,Y -486.790,Z 275.909,A 0.000,B 0.000,C 90.000,E1 199.631} C_DIS
LIN {X 0.144,Y -483.108,Z 275.897,A 0.000,B 0.000,C 90.000,E1 197.457} C_DIS
LIN {X -0.158,Y -481.168,Z 275.890,A 0.000,B 0.000,C 90.000,E1 196.260} C_DIS
LIN {X -0.050,Y -477.486,Z 275.877,A 0.000,B 0.000,C 90.000,E1 193.772} C_DIS
LIN {X -0.008,Y -474.712,Z 275.864,A 0.000,B 0.000,C 90.000,E1 191.591} C_DIS
LIN {X 0.223,Y -472.009,Z 275.852,A 0.000,B 0.000,C 90.000,E1 189.378} C_DIS
LIN {X -0.226,Y -469.711,Z 275.840,A 0.000,B 0.000,C 90.000,E1 187.239} C_DIS
LIN {X 0.149,Y -467.570,Z 275.828,A 0.000,B 0.000,C 90.000,E1 184.992} C_DIS
LIN {X -0.063,Y -465.279,Z 275.812,A 0.000,B 0.000,C 90.000,E1 182.178} C_DIS
LIN {X 0.106,Y -463.751,Z 275.800,A 0.000,B 0.000,C 90.000,E1 179.943} C_DIS
LIN {X -0.017,Y -462.483,Z 275.786,A 0.000,B 0.000,C 90.000,E1 177.421} C_DIS
